Fanuc TP program (LS listing): makrostp.ls

/PROG  MAKROSTP
/ATTR
OWNER		= MNEDITOR;
COMMENT		= "MAKRO_SCHRITT";
PROG_SIZE	= 110862;
CREATE		= DATE 11-01-11  TIME 07:00:00;
MODIFIED	= DATE 18-04-15  TIME 10:51:52;
FILE_NAME	= ;
VERSION		= 0;
LINE_COUNT	= 4830;
MEMORY_SIZE	= 113490;
PROTECT		= READ_WRITE;
TCD:  STACK_SIZE	= 0,
      TASK_PRIORITY	= 100,
      TIME_SLICE	= 0,
      BUSY_LAMP_OFF	= 1,
      ABORT_REQUEST	= 7,
      PAUSE_REQUEST	= 3;
DEFAULT_GROUP	= *,*,*,*,*;
CONTROL_CODE	= 00000000 00000010;
/MN
   1:  !Schrittkette Konzernstandard ;
   2:  !KS24 ;
   3:  !Version: 02 ;
   4:  !Stand: 011 ;
   5:  !letzte Aenderung 22.03.2017 KN ;
   6:   ;
   7:  !Zaehler [41] = aktueller Schritt ;
   8:  !Zaehler [42] = letzter Schritt ;
   9:  R[41]=0    ;
  10:  R[42]=0    ;
  11:   ;
  12:   ;
  13:  !*********************** ;
  14:  !*********************** ;
  15:  !* Start Makro_Schritt * ;
  16:  !*********************** ;
  17:  !*********************** ;
  18:   ;
  19:   ;
  20:  !***************************** ;
  21:  !*         Schritt 1         * ;
  22:  !* E/A's / Flags Ruecksetzen * ;
  23:  !***************************** ;
  24:   ;
  25:  !Loop fuer Schrittkette LBL[1] ;
  26:  LBL[1] ;
  27:  R[41]=1    ;
  28:  !Statusbildschirm einblenden ;
  29:  DO[18181]=(OFF) ;
  30:  !SK1 KF1 KS1 KE1 ;
  31:  DO[786]=(F[830] AND DO[786]) ;
  32:  DO[722]=(!F[830] AND DO[722]) ;
  33:  DO[834]=(OFF) ;
  34:  DO[842]=(OFF) ;
  35:  DO[847]=(OFF) ;
  36:  !SK2 KF2 KS2 KE2 ;
  37:  DO[946]=(F[831] AND DO[946]) ;
  38:  DO[882]=(!F[831] AND DO[882]) ;
  39:  DO[994]=(OFF) ;
  40:  DO[995]=(OFF) ;
  41:  DO[1002]=(OFF) ;
  42:  !SK3 KF3 KS3 KE3 ;
  43:  DO[1106]=(F[832] AND DO[1106]) ;
  44:  DO[1042]=(!F[832] AND DO[1042]) ;
  45:  DO[1154]=(OFF) ;
  46:  DO[1155]=(OFF) ;
  47:  DO[1162]=(OFF) ;
  48:  !KS1 KS2 KS3 ;
  49:  DO[3969]=(OFF) ;
  50:  DO[3970]=(OFF) ;
  51:  DO[3971]=(OFF) ;
  52:  !Auswahl EZ1/SP1 an KF2 ;
  53:  F[72]=(OFF) ;
  54:  !Auswahl EZ1/SP1 an KF3 ;
  55:  F[73]=(OFF) ;
  56:  !Auswert. KF Umdrehungen EZ1/SP1 ;
  57:  F[94]=(OFF) ;
  58:  F[95]=(OFF) ;
  59:  F[96]=(OFF) ;
  60:  F[97]=(OFF) ;
  61:  F[98]=(OFF) ;
  62:  F[99]=(OFF) ;
  63:  F[100]=(OFF) ;
  64:  F[101]=(OFF) ;
  65:  F[102]=(OFF) ;
  66:  F[103]=(OFF) ;
  67:  F[104]=(OFF) ;
  68:  F[105]=(OFF) ;
  69:  F[106]=(OFF) ;
  70:  F[107]=(OFF) ;
  71:  F[108]=(OFF) ;
  72:  F[109]=(OFF) ;
  73:  F[110]=(OFF) ;
  74:  F[111]=(OFF) ;
  75:  F[112]=(OFF) ;
  76:  F[113]=(OFF) ;
  77:  F[114]=(OFF) ;
  78:  F[115]=(OFF) ;
  79:  F[116]=(OFF) ;
  80:  F[117]=(OFF) ;
  81:  !Auswert. KF Umdrehungen EZ2/SP2 ;
  82:  F[150]=(OFF) ;
  83:  F[151]=(OFF) ;
  84:  F[152]=(OFF) ;
  85:  F[153]=(OFF) ;
  86:  F[154]=(OFF) ;
  87:  F[155]=(OFF) ;
  88:  !Auswert. KF Umdrehungen EZ3/SP3 ;
  89:  F[186]=(OFF) ;
  90:  F[187]=(OFF) ;
  91:  F[188]=(OFF) ;
  92:  F[189]=(OFF) ;
  93:  F[190]=(OFF) ;
  94:  F[191]=(OFF) ;
  95:  !Hilfsflags beim Fraesen ;
  96:  F[287]=(OFF) ;
  97:  F[290]=(OFF) ;
  98:  F[291]=(OFF) ;
  99:  F[301]=(OFF) ;
 100:  !Hilfsflags SZ2 an SK1 ;
 101:  F[307]=(OFF) ;
 102:  F[308]=(OFF) ;
 103:  !Hilfsflags KF Initiator ;
 104:  F[312]=(OFF) ;
 105:  F[313]=(OFF) ;
 106:  !RSK Fehlerausgaben ;
 107:  F[322]=(OFF) ;
 108:  F[323]=(OFF) ;
 109:  F[324]=(OFF) ;
 110:  F[325]=(OFF) ;
 111:  F[326]=(OFF) ;
 112:  F[327]=(OFF) ;
 113:  F[328]=(OFF) ;
 114:  F[329]=(OFF) ;
 115:  !Flag KL1 Spueleimer ;
 116:  F[352]=(OFF) ;
 117:  F[353]=(OFF) ;
 118:  !Flag KL2 Spueleimer ;
 119:  F[373]=(OFF) ;
 120:  F[374]=(OFF) ;
 121:  !Flag KL3 Spueleimer ;
 122:  F[394]=(OFF) ;
 123:  F[395]=(OFF) ;
 124:  !Flag MS Reinigung gestartet ;
 125:  F[604]=(OFF) ;
 126:  F[605]=(OFF) ;
 127:  F[608]=(OFF) ;
 128:  !Flag für Grundstellung RSK ;
 129:  F[321]=(OFF) ;
 130:  !Ruecksetzen Fraeszaehler ;
 131:  R[1]=0    ;
 132:  R[42]=1    ;
 133:  JMP LBL[2] ;
 134:   ;
 135:   ;
 136:  !************************ ;
 137:  !************************ ;
 138:  !* RSK in Grundstellung * ;
 139:  !************************ ;
 140:  !************************ ;
 141:   ;
 142:   ;
 143:  !*********************** ;
 144:  !*      Schritt 2      * ;
 145:  !* Funktionsauswertung * ;
 146:  !*********************** ;
 147:   ;
 148:  LBL[2] ;
 149:  R[41]=2    ;
 150:  F[321]=(ON) ;
 151:   ;
 152:  !Fraesen ROB EZ1/SP1 SZ1-SZ4 ;
 153:  !an KF1 ;
 154:  IF ((F[90] AND !F[91]) AND !F[72] AND !F[73] AND !F[565] AND (F[64] OR F[65] OR F[66] OR F[67])),R[41]=3 ;
 155:   ;
 156:  !Fraesen ROB EZ1/SP1 SZ1-SZ4 ;
 157:  !an KF2 ;
 158:  IF ((F[90] AND !F[91]) AND F[72] AND !F[73] AND !F[565] AND (F[64] OR F[65] OR F[66] OR F[67])),R[41]=58 ;
 159:   ;
 160:  !Fraesen ROB EZ1/SP1 SZ1-SZ4 ;
 161:  !an KF3 ;
 162:  IF ((F[90] AND !F[91]) AND !F[72] AND F[73] AND !F[565] AND (F[64] OR F[65] OR F[66] OR F[67])),R[41]=64 ;
 163:   ;
 164:  !Fraesen STAT EZ1/SP1 ;
 165:  IF (F[92] AND !F[93]),R[41]=9 ;
 166:   ;
 167:  !Fraesen STAT EZ2/SP2 ;
 168:  IF (F[148] AND !F[149]),R[41]=18 ;
 169:   ;
 170:  !Fraesen STAT EZ3/SP3 ;
 171:  IF (F[184] AND !F[185]),R[41]=27 ;
 172:   ;
 173:  !MS1 Reinigung an KS3 ;
 174:  IF (F[603] AND !F[605] AND F[528] AND !F[529]),R[41]=36 ;
 175:   ;
 176:  !MS2 Reinigung an KS2 ;
 177:  IF (F[607] AND !F[609] AND F[528] AND !F[529]),R[41]=40 ;
 178:   ;
 179:  !KL1 Spueleimer (an Pneum. Schwen ;
 180:  !in Arbeitsstellung schwenken ;
 181:  IF (!F[352] AND F[353] AND !F[355] AND ((F[523] AND !F[524]) OR (!F[523] AND F[524]))),R[41]=44 ;
 182:   ;
 183:  !KL1 Spueleimer (an Pneum. Schwen ;
 184:  !in Ruhestellung schwenken ;
 185:  IF (F[352] AND !F[353] AND !F[355] AND ((F[523] AND !F[524]) OR (!F[523] AND F[524]))),R[41]=45 ;
 186:   ;
 187:  !KL2 Spueleimer (an Pneum. Schwen ;
 188:  !in Arbeitsstellung schwenken ;
 189:  IF (!F[373] AND F[374] AND !F[376] AND ((F[523] AND !F[524]) OR (!F[523] AND F[524]))),R[41]=46 ;
 190:   ;
 191:  !KL2 Spueleimer (an Pneum. Schwen ;
 192:  !in Ruhestellung schwenken ;
 193:  IF (F[373] AND !F[374] AND !F[376] AND ((F[523] AND !F[524]) OR (!F[523] AND F[524]))),R[41]=47 ;
 194:   ;
 195:  !KL3 Spueleimer (an Pneum. Schwen ;
 196:  !in Arbeitsstellung schwenken ;
 197:  IF (!F[394] AND F[395] AND !F[397] AND ((F[523] AND !F[524]) OR (!F[523] AND F[524]))),R[41]=48 ;
 198:   ;
 199:  !KL3 Spueleimer (an Pneum. Schwen ;
 200:  !in Ruhestellung schwenken ;
 201:  IF (F[394] AND !F[395] AND !F[397] AND ((F[523] AND !F[524]) OR (!F[523] AND F[524]))),R[41]=49 ;
 202:   ;
 203:  !MS1 Reinigung (an Pneum. Schwenk ;
 204:  IF (F[603] AND !F[605] AND !F[528] AND F[529]),R[41]=50 ;
 205:   ;
 206:  !Fraesen ROB STP SZ1 ;
 207:  IF (F[64] AND !F[65] AND !F[66] AND !F[67] AND F[90] AND !F[91] AND F[565] AND !F[805]),R[41]=70 ;
 208:   ;
 209:  !Fraesen ROB STP SZ1 mit Kappenw. ;
 210:  IF (F[64] AND !F[65] AND !F[66] AND !F[67] AND F[90] AND !F[91] AND F[565] AND F[805]),R[41]=76 ;
 211:   ;
 212:  !Warte Zeit für CPU ;
 213:  WAIT    .20(sec) ;
 214:   ;
 215:  R[42]=2    ;
 216:  JMP LBL[R[41]] ;
 217:   ;
 218:   ;
 219:  !*************************** ;
 220:  !*************************** ;
 221:  !* Fraesen Rob EZ1 SZ1-SZ4 * ;
 222:  !*          an KF1         * ;
 223:  !*************************** ;
 224:  !*************************** ;
 225:   ;
 226:   ;
 227:  !**************************** ;
 228:  !*        Schritt 3         * ;
 229:  !* Rob EZ1 SZ1-SZ4 Auswert. * ;
 230:  !**************************** ;
 231:   ;
 232:  LBL[3] ;
 233:  R[41]=3    ;
 234:  !RSK gestartet ;
 235:  F[321]=(OFF) ;
 236:  GO[1]=(31) ;
 237:  IF (F[64]),GO[3]=(31) ;
 238:  IF (F[65]),GO[3]=(32) ;
 239:  IF (F[66]),GO[3]=(33) ;
 240:  IF (F[67]),GO[3]=(34) ;
 241:  WAIT    .10(sec) ;
 242:  DO[116]=(ON) ;
 243:  DO[130]=(ON) ;
 244:  DO[718]=(OFF) ;
 245:  DO[717]=(!DI[717]) ;
 246:  DO[18181]=(ON) ;
 247:  WAIT (DI[717])    ;
 248:  DO[18181]=(OFF) ;
 249:  DO[717]=(OFF) ;
 250:  !Anwahl Startfraesen ;
 251:  IF (F[90] AND F[78] AND !F[79]),R[41]=4 ;
 252:  !Anwahl Normalfraesen ;
 253:  IF (F[90] AND !F[78] AND F[79]),R[41]=6 ;
 254:  R[42]=3    ;
 255:  JMP LBL[R[41]] ;
 256:   ;
 257:  !***************************** ;
 258:  !*         Schritt 4         * ;
 259:  !* Rob EZ1 SZ1-SZ4 SF Teil 1 * ;
 260:  !***************************** ;
 261:   ;
 262:  LBL[4] ;
 263:  R[41]=4    ;
 264:  !RSK gestartet ;
 265:  F[321]=(OFF) ;
 266:  F[329]=(OFF) ;
 267:  F[325]=(OFF) ;
 268:  DO[718]=(OFF) ;
 269:  DO[717]=(!DI[717]) ;
 270:  DO[18181]=(ON) ;
 271:  WAIT (DI[717])    ;
 272:  DO[18181]=(OFF) ;
 273:  DO[834]=(ON) ;
 274:  DO[858]=(ON) ;
 275:  DO[835]=(F[330]) ;
 276:  DO[859]=(F[330]) ;
 277:  DO[717]=(OFF) ;
 278:  !Warte Fraeser laeuft ;
 279:  TIMER[7]=((-3)) ;
 280:  WAIT ((!DI[834] AND !F[289]) OR (!DI[858] AND F[289]) OR (TIMER[7]>=0))    ;
 281:  WAIT ((DI[834] AND !F[289]) OR (DI[858] AND F[289]) OR (TIMER[7]>=0))    ;
 282:  F[322]=((TIMER[7]>=0)) ;
 283:  DO[18181]=(ON) ;
 284:  WAIT ((!DI[834] AND !F[289]) OR (!DI[858] AND F[289]))    ;
 285:  WAIT ((DI[834] AND !F[289]) OR (DI[858] AND F[289]))    ;
 286:  DO[18181]=(OFF) ;
 287:  F[322]=(OFF) ;
 288:  !EZ1/SP1 schliessen ;
 289:  DO[718]=(ON) ;
 290:  TIMER[9]=((-4)) ;
 291:  !EZ1/SP1 Kraft erreicht ;
 292:  WAIT ((DI[718] AND !DI[772] AND !DI[780] AND !DI[774] AND !DI[775]) OR (TIMER[9]>=0))    ;
 293:  DO[18181]=(ON) ;
 294:  DO[718]=((TIMER[9]<0)) ;
 295:  DO[834]=((TIMER[9]<0)) ;
 296:  DO[858]=((TIMER[9]<0)) ;
 297:  WAIT ((DI[718] AND !DI[772] AND !DI[780] AND !DI[774] AND !DI[775]) OR DI[26] OR DI[27])    ;
 298:  F[325]=(DI[26] OR DI[27]) ;
 299:  DO[18181]=(OFF) ;
 300:  !EZ1/SP1 Fehler Kraftaufbau ;
 301:  IF (F[325]),JMP LBL[406] ;
 302:  TIMER[9]=((-5)) ;
 303:  LBL[400] ;
 304:  WAIT ((!DI[834] AND !F[289]) OR (!DI[858] AND F[289]) OR F[325] OR (TIMER[9]>=0))    ;
 305:  WAIT ((DI[834] AND !F[289]) OR (DI[858] AND F[289]) OR F[325] OR (TIMER[9]>=0))    ;
 306:  R[1]=(R[1]+1) ;
 307:  F[329]=((TIMER[9]>=0)) ;
 308:  !Fraeszeit ueberschritten ;
 309:  IF (F[329]),JMP LBL[406] ;
 310:  IF (F[64]),JMP LBL[402] ;
 311:  IF (F[65]),JMP LBL[403] ;
 312:  IF (F[66]),JMP LBL[404] ;
 313:  IF (F[67]),JMP LBL[405] ;
 314:  !Umdrehungen Vergl.SZ1 ;
 315:  LBL[402] ;
 316:  !Umdrehungen Vergleichen ;
 317:  IF (R[1]<R[2]),JMP LBL[400] ;
 318:  JMP LBL[401] ;
 319:  !Umdrehungen Vergl.SZ2 ;
 320:  LBL[403] ;
 321:  !Umdrehungen Vergleichen ;
 322:  IF (R[1]<R[8]),JMP LBL[400] ;
 323:  JMP LBL[401] ;
 324:  !Umdrehungen Vergl.SZ3 ;
 325:  LBL[404] ;
 326:  !Umdrehungen Vergleichen ;
 327:  IF (R[1]<R[11]),JMP LBL[400] ;
 328:  JMP LBL[401] ;
 329:  !Umdrehungen Vergl.SZ4 ;
 330:  LBL[405] ;
 331:  !Umdrehungen Vergleichen ;
 332:  IF (R[1]<R[14]),JMP LBL[400] ;
 333:  JMP LBL[401] ;
 334:  LBL[401] ;
 335:  IF (F[64]),F[94]=(ON) ;
 336:  IF (F[65]),F[100]=(ON) ;
 337:  IF (F[66]),F[106]=(ON) ;
 338:  IF (F[67]),F[112]=(ON) ;
 339:  LBL[406] ;
 340:  DO[834]=((TIMER[9]<0)) ;
 341:  DO[858]=((TIMER[9]<0)) ;
 342:  !Fraeser ausblasen EIN ;
 343:  DO[835]=(F[330] OR (TIMER[9]<0)) ;
 344:  DO[859]=(F[330] OR (TIMER[9]<0)) ;
 345:  DO[718]=(OFF) ;
 346:  !EZ1/SP1 oeffnen ;
 347:  DO[717]=(!DI[717]) ;
 348:  DO[18181]=(F[329]) ;
 349:  WAIT (!F[329] OR DI[26] OR DI[27])    ;
 350:  DO[18181]=(OFF) ;
 351:  DO[18181]=(ON) ;
 352:  WAIT (DI[717])    ;
 353:  DO[18181]=(OFF) ;
 354:  DO[717]=(OFF) ;
 355:  !Umdrehungen ruecksetzen ;
 356:  R[1]=0    ;
 357:  R[42]=4    ;
 358:  IF (F[329] OR F[325]),JMP LBL[4] ;
 359:  JMP LBL[5] ;
 360:   ;
 361:  !***************************** ;
 362:  !*         Schritt 5         * ;
 363:  !* Rob EZ1 SZ1-SZ4 SF Teil 2 * ;
 364:  !***************************** ;
 365:   ;
 366:  LBL[5] ;
 367:  R[41]=5    ;
 368:  !RSK gestartet ;
 369:  F[321]=(OFF) ;
 370:  F[329]=(OFF) ;
 371:  F[325]=(OFF) ;
 372:  DO[718]=(OFF) ;
 373:  DO[717]=(!DI[717]) ;
 374:  DO[18181]=(ON) ;
 375:  WAIT (DI[717])    ;
 376:  DO[18181]=(OFF) ;
 377:  DO[834]=(ON) ;
 378:  DO[858]=(ON) ;
 379:  DO[717]=(OFF) ;
 380:  !EZ1/SP1 schliessen ;
 381:  DO[718]=(ON) ;
 382:  !Fraeser ausblasen AUS/AN ;
 383:  DO[835]=(F[330]) ;
 384:  DO[859]=(F[330]) ;
 385:  TIMER[9]=((-4)) ;
 386:  !EZ1/SP1 Kraft erreicht ;
 387:  WAIT ((DI[718] AND !DI[772] AND !DI[780] AND !DI[774] AND !DI[775]) OR (TIMER[9]>=0))    ;
 388:  DO[18181]=(ON) ;
 389:  DO[718]=((TIMER[9]<0)) ;
 390:  DO[834]=((TIMER[9]<0)) ;
 391:  DO[858]=((TIMER[9]<0)) ;
 392:  WAIT ((DI[718] AND !DI[772] AND !DI[780] AND !DI[774] AND !DI[775]) OR DI[26] OR DI[27])    ;
 393:  F[325]=(DI[26] OR DI[27]) ;
 394:  DO[18181]=(OFF) ;
 395:  !EZ1/SP1 Fehler Kraftaufbau ;
 396:  IF (F[325]),JMP LBL[5] ;
 397:  TIMER[9]=((-5)) ;
 398:  LBL[500] ;
 399:  WAIT ((!DI[834] AND !F[289]) OR (!DI[858] AND F[289]) OR F[325] OR (TIMER[9]>=0))    ;
 400:  WAIT ((DI[834] AND !F[289]) OR (DI[858] AND F[289]) OR F[325] OR (TIMER[9]>=0))    ;
 401:  R[1]=(R[1]+1) ;
 402:  F[329]=((TIMER[9]>=0)) ;
 403:  !Fraeszeit ueberschritten ;
 404:  IF (F[329]),JMP LBL[506] ;
 405:  IF (F[64]),JMP LBL[502] ;
 406:  IF (F[65]),JMP LBL[503] ;
 407:  IF (F[66]),JMP LBL[504] ;
 408:  IF (F[67]),JMP LBL[505] ;
 409:  !Umdrehungen Vergl.SZ1 ;
 410:  LBL[502] ;
 411:  !Umdrehungen Vergleichen ;
 412:  IF (R[1]<R[3]),JMP LBL[500] ;
 413:  JMP LBL[501] ;
 414:  !Umdrehungen Vergl.SZ2 ;
 415:  LBL[503] ;
 416:  !Umdrehungen Vergleichen ;
 417:  IF (R[1]<R[9]),JMP LBL[500] ;
 418:  JMP LBL[501] ;
 419:  !Umdrehungen Vergl.SZ3 ;
 420:  LBL[504] ;
 421:  !Umdrehungen Vergleichen ;
 422:  IF (R[1]<R[12]),JMP LBL[500] ;
 423:  JMP LBL[501] ;
 424:  !Umdrehungen Vergl.SZ4 ;
 425:  LBL[505] ;
 426:  !Umdrehungen Vergleichen ;
 427:  IF (R[1]<R[15]),JMP LBL[500] ;
 428:  JMP LBL[501] ;
 429:  LBL[501] ;
 430:  IF (F[64]),F[96]=(ON) ;
 431:  IF (F[65]),F[102]=(ON) ;
 432:  IF (F[66]),F[108]=(ON) ;
 433:  IF (F[67]),F[114]=(ON) ;
 434:  LBL[506] ;
 435:  DO[834]=((TIMER[9]<0)) ;
 436:  DO[858]=((TIMER[9]<0)) ;
 437:  !Fraeser ausblasen EIN ;
 438:  DO[835]=PULSE,4.0sec ;
 439:  DO[859]=PULSE,4.0sec ;
 440:  DO[718]=(OFF) ;
 441:  !EZ1/SP1 oeffnen ;
 442:  DO[717]=(!DI[717]) ;
 443:  DO[18181]=(F[329]) ;
 444:  WAIT (!F[329] OR DI[26] OR DI[27])    ;
 445:  DO[18181]=(OFF) ;
 446:  DO[18181]=(ON) ;
 447:  WAIT (DI[717])    ;
 448:  DO[18181]=(OFF) ;
 449:  DO[717]=(OFF) ;
 450:  !Umdrehungen ruecksetzen ;
 451:  R[1]=0    ;
 452:  R[42]=5    ;
 453:  IF (F[329] OR F[325]),JMP LBL[5] ;
 454:  JMP LBL[7] ;
 455:   ;
 456:  !********************** ;
 457:  !*     Schritt 6      * ;
 458:  !* Rob EZ1 SZ1-SZ4 NF * ;
 459:  !********************** ;
 460:   ;
 461:  LBL[6] ;
 462:  R[41]=6    ;
 463:  !RSK gestartet ;
 464:  F[321]=(OFF) ;
 465:  F[329]=(OFF) ;
 466:  F[325]=(OFF) ;
 467:  !Zähler wegspeichern für 2ten Hub ;
 468:  R[45]=(R[4]) ;
 469:  IF (F[98] AND F[732]),R[4]=(R[43]) ;
 470:  !Überprüfungung Zangenstellung ;
 471:  DO[718]=(OFF) ;
 472:  DO[717]=(!DI[717]) ;
 473:  DO[18181]=(ON) ;
 474:  WAIT (DI[717])    ;
 475:  DO[18181]=(OFF) ;
 476:  DO[834]=(ON) ;
 477:  DO[835]=(F[330]) ;
 478:  DO[858]=(ON) ;
 479:  DO[859]=(F[330]) ;
 480:  DO[717]=(OFF) ;
 481:  !Warte Fraeser laeuft ;
 482:  TIMER[7]=((-3)) ;
 483:  WAIT ((!DI[834] AND !F[289]) OR (!DI[858] AND F[289]) OR (TIMER[7]>=0))    ;
 484:  WAIT ((DI[834] AND !F[289]) OR (DI[858] AND F[289]) OR (TIMER[7]>=0))    ;
 485:  F[322]=((TIMER[7]>=0)) ;
 486:  DO[18181]=(ON) ;
 487:  WAIT ((!DI[834] AND !F[289]) OR (!DI[858] AND F[289]))    ;
 488:  WAIT ((DI[834] AND !F[289]) OR (DI[858] AND F[289]))    ;
 489:  DO[18181]=(OFF) ;
 490:  F[322]=(OFF) ;
 491:  !EZ1/SP1 schliessen ;
 492:  DO[718]=(ON) ;
 493:  TIMER[9]=((-4)) ;
 494:  !EZ1/SP1 Kraft erreicht ;
 495:  WAIT ((DI[718] AND !DI[772] AND !DI[780] AND !DI[774] AND !DI[775]) OR (TIMER[9]>=0))    ;
 496:  DO[18181]=(ON) ;
 497:  DO[718]=((TIMER[9]<0)) ;
 498:  DO[834]=((TIMER[9]<0)) ;
 499:  DO[858]=((TIMER[9]<0)) ;
 500:  WAIT ((DI[718] AND !DI[772] AND !DI[780] AND !DI[774] AND !DI[775]) OR DI[26] OR DI[27])    ;
 501:  F[325]=(DI[26] OR DI[27]) ;
 502:  DO[18181]=(OFF) ;
 503:  !EZ1/SP1 Fehler Kraftaufbau ;
 504:  IF (F[325]),JMP LBL[6] ;
 505:  TIMER[9]=((-5)) ;
 506:  LBL[600] ;
 507:  WAIT ((!DI[834] AND !F[289]) OR (!DI[858] AND F[289]) OR F[325] OR (TIMER[9]>=0))    ;
 508:  WAIT ((DI[834] AND !F[289]) OR (DI[858] AND F[289]) OR F[325] OR (TIMER[9]>=0))    ;
 509:  R[1]=(R[1]+1) ;
 510:  F[329]=((TIMER[9]>=0)) ;
 511:  !Fraeszeit ueberschritten ;
 512:  IF (F[329]),JMP LBL[606] ;
 513:  IF (F[64]),JMP LBL[602] ;
 514:  IF (F[65]),JMP LBL[603] ;
 515:  IF (F[66]),JMP LBL[604] ;
 516:  IF (F[67]),JMP LBL[605] ;
 517:  !Umdrehungen Vergl.SZ1 ;
 518:  LBL[602] ;
 519:  !Umdrehungen Vergleichen ;
 520:  IF (R[1]<R[4]),JMP LBL[600] ;
 521:  JMP LBL[601] ;
 522:  !Umdrehungen Vergl.SZ2 ;
 523:  LBL[603] ;
 524:  !Umdrehungen Vergleichen ;
 525:  IF (R[1]<R[10]),JMP LBL[600] ;
 526:  !Umdrehungen Vergl.SZ3 ;
 527:  LBL[604] ;
 528:  !Umdrehungen Vergleichen ;
 529:  IF (R[1]<R[13]),JMP LBL[600] ;
 530:  JMP LBL[601] ;
 531:  !Umdrehungen Vergl.SZ4 ;
 532:  LBL[605] ;
 533:  !Umdrehungen Vergleichen ;
 534:  IF (R[1]<R[16]),JMP LBL[600] ;
 535:  LBL[601] ;
 536:  !EZ1/SP1 2 Huebe bei NF ;
 537:  IF (!F[130]),JMP LBL[606] ;
 538:  IF (F[98]),F[96]=(ON) ;
 539:  IF (F[104]),F[96]=(ON) ;
 540:  IF (F[110]),F[96]=(ON) ;
 541:  IF (F[116]),F[96]=(ON) ;
 542:  IF (F[64]),F[98]=(ON) ;
 543:  IF (F[65]),F[104]=(ON) ;
 544:  IF (F[66]),F[110]=(ON) ;
 545:  IF (F[67]),F[116]=(ON) ;
 546:  LBL[606] ;
 547:  DO[834]=((TIMER[9]<0)) ;
 548:  DO[858]=((TIMER[9]<0)) ;
 549:  !Fraeser ausblasen EIN ;
 550:  DO[835]=PULSE,4.0sec ;
 551:  DO[859]=PULSE,4.0sec ;
 552:  DO[718]=(OFF) ;
 553:  !EZ1/SP1 oeffnen ;
 554:  DO[717]=(!DI[717]) ;
 555:  DO[18181]=(F[329]) ;
 556:  WAIT (!F[329] OR DI[26] OR DI[27])    ;
 557:  DO[18181]=(OFF) ;
 558:  DO[18181]=(ON) ;
 559:  WAIT (DI[717])    ;
 560:  DO[18181]=(OFF) ;
 561:  DO[717]=(OFF) ;
 562:  !Umdrehungen ruecksetzen ;
 563:  R[1]=0    ;
 564:  R[42]=6    ;
 565:  !Zähler umschreiben für 2ten Hub ;
 566:  IF (F[98] AND F[732] AND F[64]),GO[3]=36 ;
 567:  IF (F[104] AND F[732] AND F[65]),GO[3]=37 ;
 568:  IF (F[110] AND F[732] AND F[66]),GO[3]=38 ;
 569:  IF (F[116] AND F[732] AND F[67]),GO[3]=39 ;
 570:  IF (F[96] AND F[732]),R[4]=(R[45]) ;
 571:  !Aufruf 2ter Hub ;
 572:  IF (F[329] OR (!F[96] AND F[130])),JMP LBL[6] ;
 573:  IF (F[64]),F[98]=(ON) ;
 574:  IF (F[65]),F[104]=(ON) ;
 575:  IF (F[66]),F[110]=(ON) ;
 576:  IF (F[67]),F[116]=(ON) ;
 577:  JMP LBL[7] ;
 578:   ;
 579:  !******************************* ;
 580:  !*         Schritt 7           * ;
 581:  !* Rob EZ1 SZ1-SZ4 i.O./n.i.O. * ;
 582:  !******************************* ;
 583:   ;
 584:  LBL[7] ;
 585:  R[41]=7    ;
 586:  !Fraesueberwachung starten ;
 587:  IF (F[64]),JMP LBL[701] ;
 588:  IF (F[65]),JMP LBL[702] ;
 589:  IF (F[66]),JMP LBL[703] ;
 590:  IF (F[67]),JMP LBL[704] ;
 591:  LBL[701] ;
 592:  TIMER[7]=((-3)) ;
 593:  WAIT (F[64] AND ((F[79] AND F[98]) OR (F[78] AND F[94] AND F[96])) OR (TIMER[7]>=0))    ;
 594:  F[329]=((TIMER[7]>=0)) ;
 595:  DO[18181]=(ON) ;
 596:  WAIT (F[64] AND ((F[79] AND F[98]) OR (F[78] AND F[94] AND F[96])))    ;
 597:  DO[18181]=(OFF) ;
 598:  JMP LBL[700] ;
 599:  LBL[702] ;
 600:  TIMER[7]=((-3)) ;
 601:  WAIT (F[65] AND ((F[79] AND F[104]) OR (F[78] AND F[100] AND F[102])) OR (TIMER[7]>=0))    ;
 602:  F[329]=((TIMER[7]>=0)) ;
 603:  DO[18181]=(ON) ;
 604:  WAIT (F[65] AND ((F[79] AND F[104]) OR (F[78] AND F[100] AND F[102])))    ;
 605:  DO[18181]=(OFF) ;
 606:  JMP LBL[700] ;
 607:  LBL[703] ;
 608:  TIMER[7]=((-3)) ;
 609:  WAIT (F[66] AND ((F[79] AND F[110]) OR (F[78] AND F[106] AND F[108])) OR (TIMER[7]>=0))    ;
 610:  F[329]=((TIMER[7]>=0)) ;
 611:  DO[18181]=(ON) ;
 612:  WAIT (F[66] AND ((F[79] AND F[110]) OR (F[78] AND F[106] AND F[108])))    ;
 613:  DO[18181]=(OFF) ;
 614:  JMP LBL[700] ;
 615:  LBL[704] ;
 616:  TIMER[7]=((-3)) ;
 617:  WAIT (F[67] AND ((F[79] AND F[116]) OR (F[78] AND F[112] AND F[114])) OR (TIMER[7]>=0))    ;
 618:  F[329]=((TIMER[7]>=0)) ;
 619:  DO[18181]=(ON) ;
 620:  WAIT (F[67] AND ((F[79] AND F[116]) OR (F[78] AND F[112] AND F[114])))    ;
 621:  DO[18181]=(OFF) ;
 622:  JMP LBL[700] ;
 623:  LBL[700] ;
 624:  R[41]=8    ;
 625:  !KF1 U-Merker ruecksetzen ;
 626:  F[94]=(OFF) ;
 627:  F[96]=(OFF) ;
 628:  F[98]=(OFF) ;
 629:  F[100]=(OFF) ;
 630:  F[102]=(OFF) ;
 631:  F[104]=(OFF) ;
 632:  F[106]=(OFF) ;
 633:  F[108]=(OFF) ;
 634:  F[110]=(OFF) ;
 635:  F[112]=(OFF) ;
 636:  F[114]=(OFF) ;
 637:  F[116]=(OFF) ;
 638:  R[42]=7    ;
 639:  JMP LBL[R[41]] ;
 640:   ;
 641:  !***************************** ;
 642:  !*        Schritt 8          * ;
 643:  !* Rob EZ1 SZ1-SZ4 Quitt SK1 * ;
 644:  !* Rob EZ1 SZ1-SZ4 Quitt KE1 * ;
 645:  !***************************** ;
 646:   ;
 647:  LBL[8] ;
 648:  R[41]=8    ;
 649:  !RSK gestartet ;
 650:  F[321]=(OFF) ;
 651:  IF (F[64]),GO[3]=1 ;
 652:  IF (F[65]),GO[3]=2 ;
 653:  IF (F[66]),GO[3]=3 ;
 654:  IF (F[67]),GO[3]=4 ;
 655:  WAIT    .10(sec) ;
 656:  DO[786]=(!F[830]) ;
 657:  DO[722]=(F[830]) ;
 658:  DO[116]=(OFF) ;
 659:  DO[130]=(OFF) ;
 660:  DO[18181]=(ON) ;
 661:  WAIT ((!DI[786] AND DI[787] AND !DI[788]) OR F[830])    ;
 662:  WAIT ((!DI[722] AND DI[724] AND !DI[723] OR F[329]) OR !F[830])    ;
 663:  !FK Fraesen ;
 664:  F[91]=((!DI[786] AND DI[787] AND !DI[788] AND !F[830]) OR (!DI[722] AND DI[724] AND !DI[723] AND F[830]) AND !F[322] AND !F[325] AND !F[329]) ;
 665:  DO[18181]=(OFF) ;
 666:  DO[786]=(F[830] AND DO[786]) ;
 667:  DO[722]=(!F[830] AND DO[722]) ;
 668:  R[42]=8    ;
 669:  JMP LBL[1] ;
 670:   ;
 671:   ;
 672:  !************************ ;
 673:  !************************ ;
 674:  !* Fraesen STAT EZ1/SP1 * ;
 675:  !************************ ;
 676:  !************************ ;
 677:   ;
 678:   ;
 679:  !****************************** ;
 680:  !*         Schritt 9          * ;
 681:  !*        STAT EZ1/SP1        * ;
 682:  !* KS1 in Arbeitsst.schwenken * ;
 683:  !****************************** ;
 684:   ;
 685:  LBL[9] ;
 686:  R[41]=9    ;
 687:  !RSK gestartet ;
 688:  F[321]=(OFF) ;
 689:  GO[1]=(31) ;
 690:  GO[3]=(31) ;
 691:  WAIT    .10(sec) ;
 692:  DO[758]=(F[78]) ;
 693:  DO[759]=(F[79]) ;
 694:  DO[116]=(ON) ;
 695:  DO[130]=(ON) ;
 696:  DO[718]=(OFF) ;
 697:  DO[717]=(!DI[717]) ;
 698:  DO[18181]=(ON) ;
 699:  WAIT (DI[717])    ;
 700:  DO[18181]=(OFF) ;
 701:  DO[717]=(OFF) ;
 702:  !Ueberwachungszeit Grundstellung ;
 703:  TIMER[8]=((-4)) ;
 704:  WAIT ((DI[842] AND !DI[843] AND !DI[844] AND DI[845]) OR (TIMER[8]>=0))    ;
 705:  F[323]=((TIMER[8]>=0)) ;
 706:  DO[18181]=((TIMER[8]>=0)) ;
 707:  WAIT (DI[842] AND !DI[843] AND !DI[844] AND DI[845])    ;
 708:  DO[18181]=(OFF) ;
 709:  F[323]=(OFF) ;
 710:  TIMER[8]=((-4)) ;
 711:  DO[835]=(F[564]) ;
 712:  WAIT ((DI[835] AND F[564]) OR (!DI[835] AND !F[564]) OR (TIMER[8]>=0))    ;
 713:  F[323]=((TIMER[8]>=0)) ;
 714:  DO[18181]=((TIMER[8]>=0)) ;
 715:  WAIT ((DI[835] AND F[564]) OR (!DI[835] AND !F[564]))    ;
 716:  DO[18181]=(OFF) ;
 717:  F[323]=(OFF) ;
 718:  !Ueberwachungszeit KS1 Schwenken ;
 719:  TIMER[8]=((-6)) ;
 720:  !KS1 in Arbeitst. schwenken ;
 721:  DO[3972]=(ON) ;
 722:  WAIT (DI[841] OR (TIMER[8]>=0))    ;
 723:  DO[18181]=((TIMER[8]>=0)) ;
 724:  WAIT (DI[841])    ;
 725:  TIMER[8]=((-6)) ;
 726:  DO[18181]=(OFF) ;
 727:  WAIT ((!DI[842] AND DI[843] AND DI[844] AND !DI[845]) OR (TIMER[8]>=0))    ;
 728:  F[324]=((TIMER[8]>=0)) ;
 729:  DO[3972]=(OFF) ;
 730:  DO[18181]=((TIMER[8]>=0)) ;
 731:  WAIT ((!DI[842] AND DI[843] AND DI[844] AND !DI[845]) OR DI[26])    ;
 732:  DO[18181]=(OFF) ;
 733:  F[324]=(OFF) ;
 734:  !Sprung zurueck bei KS1 Fehler ;
 735:  IF (TIMER[8]>=0),JMP LBL[9] ;
 736:  DO[835]=(OFF) ;
 737:  TIMER[11]=((R[24])) ;
 738:  WAIT ((TIMER[11]>=0) OR !F[564])    ;
 739:  TIMER[11]=STOP ;
 740:  DO[18181]=(ON) ;
 741:  WAIT ((F[92] AND F[78]) OR (F[92] AND F[79]))    ;
 742:  DO[18181]=(OFF) ;
 743:  !Anwahl Startfraesen ;
 744:  IF (!DI[842] AND DI[843] AND F[92] AND F[78] AND !F[301]),R[41]=10 ;
 745:  !Anwahl Normalfraesen ;
 746:  IF (!DI[842] AND DI[843] AND F[92] AND (F[79] OR F[301])),R[41]=12 ;
 747:  R[42]=9    ;
 748:  JMP LBL[R[41]] ;
 749:   ;
 750:  !************************** ;
 751:  !*       Schritt 10       * ;
 752:  !* STAT EZ1/SP1 SF Teil 1 * ;
 753:  !************************** ;
 754:   ;
 755:  LBL[10] ;
 756:  R[41]=10    ;
 757:  !RSK gestartet ;
 758:  F[321]=(OFF) ;
 759:  F[329]=(OFF) ;
 760:  F[325]=(OFF) ;
 761:  DO[718]=(OFF) ;
 762:  DO[717]=(!DI[717]) ;
 763:  DO[18181]=(ON) ;
 764:  WAIT (DI[717])    ;
 765:  DO[717]=(OFF) ;
 766:  DO[18181]=(OFF) ;
 767:  DO[834]=(ON) ;
 768:  !Warte Fraeser laeuft ;
 769:  TIMER[7]=((-3)) ;
 770:  WAIT (!DI[834] OR (TIMER[7]>=0))    ;
 771:  WAIT (DI[834] OR (TIMER[7]>=0))    ;
 772:  F[322]=((TIMER[7]>=0)) ;
 773:  DO[18181]=(ON) ;
 774:  WAIT (!DI[834])    ;
 775:  WAIT (DI[834])    ;
 776:  DO[18181]=(OFF) ;
 777:  F[322]=(OFF) ;
 778:  !EZ1/SP1 schliessen ;
 779:  DO[718]=(ON) ;
 780:  !Fraeser ausblasen AUS/EIN ;
 781:  DO[847]=(F[330]) ;
 782:  TIMER[9]=((-4)) ;
 783:  !EZ1/SP1 Kraft erreicht ;
 784:  WAIT ((DI[718] AND !DI[772] AND !DI[780] AND !DI[774] AND !DI[775]) OR (TIMER[9]>=0))    ;
 785:  F[325]=((TIMER[9]>=0)) ;
 786:  DO[18181]=(ON) ;
 787:  DO[718]=((TIMER[9]<0)) ;
 788:  DO[834]=((TIMER[9]<0)) ;
 789:  WAIT ((DI[718] AND !DI[772] AND !DI[780] AND !DI[774] AND !DI[775]) OR DI[26] OR DI[27])    ;
 790:  DO[18181]=(OFF) ;
 791:  !EZ1/SP1 Fehler Kraftaufbau ;
 792:  IF (F[325]),JMP LBL[1001] ;
 793:  TIMER[9]=((-5)) ;
 794:  LBL[1000] ;
 795:  WAIT (!DI[834] OR F[325] OR (TIMER[9]>=0))    ;
 796:  WAIT (DI[834] OR F[325] OR (TIMER[9]>=0))    ;
 797:  R[1]=(R[1]+1) ;
 798:  F[329]=((TIMER[9]>=0)) ;
 799:  !Fraeszeit ueberschritten ;
 800:  IF (F[329]),JMP LBL[1001] ;
 801:  !Umdrehungen Vergleichen ;
 802:  IF (R[1]<R[2]),JMP LBL[1000] ;
 803:  F[94]=(ON) ;
 804:  LBL[1001] ;
 805:  DO[834]=((TIMER[9]<0)) ;
 806:  !Fraeser ausblasen EIN ;
 807:  DO[847]=(F[330] OR (TIMER[9]<0)) ;
 808:  DO[718]=(OFF) ;
 809:  !EZ1/SP1 oeffnen ;
 810:  DO[717]=(!DI[717]) ;
 811:  DO[18181]=(F[329]) ;
 812:  WAIT (!F[329] OR DI[26] OR DI[27])    ;
 813:  DO[18181]=(OFF) ;
 814:  DO[18181]=(ON) ;
 815:  WAIT (DI[717])    ;
 816:  DO[18181]=(OFF) ;
 817:  DO[717]=(OFF) ;
 818:  !Umdrehungen ruecksetzen ;
 819:  R[1]=0    ;
 820:  R[42]=10    ;
 821:  IF (F[329] OR F[325]),JMP LBL[10] ;
 822:  JMP LBL[11] ;
 823:   ;
 824:  !************************** ;
 825:  !*       Schritt 11       * ;
 826:  !* STAT EZ1/SP1 SF Teil 2 * ;
 827:  !************************** ;
 828:   ;
 829:  LBL[11] ;
 830:  R[41]=11    ;
 831:  !RSK gestartet ;
 832:  F[321]=(OFF) ;
 833:  F[329]=(OFF) ;
 834:  F[325]=(OFF) ;
 835:  DO[718]=(OFF) ;
 836:  DO[717]=(!DI[717]) ;
 837:  DO[18181]=(ON) ;
 838:  WAIT (DI[717])    ;
 839:  DO[18181]=(OFF) ;
 840:  DO[834]=(ON) ;
 841:  DO[717]=(OFF) ;
 842:  !EZ1/SP1 schliessen ;
 843:  DO[718]=(ON) ;
 844:  !Fraeser ausblasen AUS/EIN ;
 845:  DO[847]=(F[330]) ;
 846:  TIMER[9]=((-4)) ;
 847:  !EZ1/SP1 Kraft erreicht ;
 848:  WAIT ((DI[718] AND !DI[772] AND !DI[780] AND !DI[774] AND !DI[775]) OR (TIMER[9]>=0))    ;
 849:  F[325]=((TIMER[9]>=0)) ;
 850:  DO[18181]=(ON) ;
 851:  DO[718]=((TIMER[9]<0)) ;
 852:  DO[834]=((TIMER[9]<0)) ;
 853:  WAIT ((DI[718] AND !DI[772] AND !DI[780] AND !DI[774] AND !DI[775]) OR DI[26] OR DI[27])    ;
 854:  DO[18181]=(OFF) ;
 855:  !EZ1/SP1 Fehler Kraftaufbau ;
 856:  IF (F[325]),JMP LBL[1101] ;
 857:  TIMER[9]=((-5)) ;
 858:  LBL[1100] ;
 859:  WAIT (!DI[834] OR F[325] OR (TIMER[9]>=0))    ;
 860:  WAIT (DI[834] OR F[325] OR (TIMER[9]>=0))    ;
 861:  R[1]=(R[1]+1) ;
 862:  F[329]=((TIMER[9]>=0)) ;
 863:  !Fraeszeit ueberschritten ;
 864:  IF (F[329]),JMP LBL[1101] ;
 865:  !Umdrehungen Vergleichen ;
 866:  IF (R[1]<R[3]),JMP LBL[1100] ;
 867:  F[96]=(ON) ;
 868:  LBL[1101] ;
 869:  DO[834]=((TIMER[9]<0)) ;
 870:  !Fraeser ausblasen EIN ;
 871:  DO[847]=PULSE,4.0sec ;
 872:  DO[718]=(OFF) ;
 873:  !EZ1/SP1 oeffnen ;
 874:  DO[717]=(!DI[717]) ;
 875:  DO[18181]=(F[329]) ;
 876:  WAIT (!F[329] OR DI[26] OR DI[27])    ;
 877:  DO[18181]=(OFF) ;
 878:  DO[18181]=(ON) ;
 879:  WAIT (DI[717])    ;
 880:  DO[18181]=(OFF) ;
 881:  DO[717]=(OFF) ;
 882:  !Umdrehungen ruecksetzen ;
 883:  R[1]=0    ;
 884:  R[42]=11    ;
 885:  IF (F[329] OR F[325]),JMP LBL[11] ;
 886:  JMP LBL[13] ;
 887:   ;
 888:  !******************* ;
 889:  !*   Schritt 12    * ;
 890:  !* STAT EZ1/SP1 NF * ;
 891:  !******************* ;
 892:   ;
 893:  LBL[12] ;
 894:  R[41]=12    ;
 895:  !RSK gestartet ;
 896:  F[321]=(OFF) ;
 897:  F[329]=(OFF) ;
 898:  F[325]=(OFF) ;
 899:  !Zähler wegspeichern für 2ten Hub ;
 900:  R[45]=(R[4]) ;
 901:  IF (F[98] AND F[732]),R[4]=(R[43]) ;
 902:  !Überprüfungung Zangenstellung ;
 903:  DO[718]=(OFF) ;
 904:  DO[717]=(!DI[717]) ;
 905:  DO[18181]=(ON) ;
 906:  WAIT (DI[717])    ;
 907:  DO[18181]=(OFF) ;
 908:  DO[834]=(ON) ;
 909:  DO[717]=(OFF) ;
 910:  !EZ1/SP1 schliessen ;
 911:  DO[718]=(ON) ;
 912:  !Fraeser ausblasen AUS/EIN ;
 913:  DO[847]=(F[330]) ;
 914:  TIMER[9]=((-4)) ;
 915:  !EZ1/SP1 Kraft erreicht ;
 916:  WAIT ((DI[718] AND !DI[772] AND !DI[780] AND !DI[774] AND !DI[775]) OR (TIMER[9]>=0))    ;
 917:  F[325]=((TIMER[9]>=0)) ;
 918:  DO[18181]=(ON) ;
 919:  DO[718]=((TIMER[9]<0)) ;
 920:  DO[834]=((TIMER[9]<0)) ;
 921:  WAIT ((DI[718] AND !DI[772] AND !DI[780] AND !DI[774] AND !DI[775]) OR DI[26] OR DI[27])    ;
 922:  DO[18181]=(OFF) ;
 923:  !EZ1/SP1 Fehler Kraftaufbau ;
 924:  IF (F[325]),JMP LBL[1201] ;
 925:  TIMER[9]=((-5)) ;
 926:  LBL[1200] ;
 927:  WAIT (!DI[834] OR F[325] OR (TIMER[9]>=0))    ;
 928:  WAIT (DI[834] OR F[325] OR (TIMER[9]>=0))    ;
 929:  R[1]=(R[1]+1) ;
 930:  F[329]=((TIMER[9]>=0)) ;
 931:  !Fraeszeit ueberschritten ;
 932:  IF (F[329]),JMP LBL[1201] ;
 933:  !Umdrehungen Vergleichen ;
 934:  IF (R[1]<R[4]),JMP LBL[1200] ;
 935:  !EZ1/SP1 2 Huebe bei NF ;
 936:  IF (!F[130]),JMP LBL[1201] ;
 937:  IF (F[98]),F[96]=(ON) ;
 938:  F[98]=(ON) ;
 939:  LBL[1201] ;
 940:  DO[834]=((TIMER[9]<0)) ;
 941:  !Fraeser ausblasen EIN ;
 942:  DO[847]=PULSE,4.0sec ;
 943:  !EZ1/SP1 oeffnen ;
 944:  DO[718]=(OFF) ;
 945:  DO[717]=(!DI[717]) ;
 946:  DO[18181]=(F[329]) ;
 947:  WAIT (!F[329] OR DI[26] OR DI[27])    ;
 948:  DO[18181]=(OFF) ;
 949:  DO[18181]=(ON) ;
 950:  WAIT (DI[717])    ;
 951:  DO[18181]=(OFF) ;
 952:  DO[717]=(OFF) ;
 953:  !Umdrehungen ruecksetzen ;
 954:  R[1]=0    ;
 955:  R[42]=12    ;
 956:  !Zähler umschreiben für 2ten Hub ;
 957:  IF (F[98] AND F[732]),GO[3]=36 ;
 958:  IF (F[96] AND F[732]),R[4]=(R[45]) ;
 959:  IF (F[329] OR F[325] OR (!F[96] AND F[130])),JMP LBL[12] ;
 960:  F[98]=(ON) ;
 961:  JMP LBL[13] ;
 962:   ;
 963:  !**************************** ;
 964:  !*        Schritt 13        * ;
 965:  !* STAT EZ1/SP1 i.O./n.i.O. * ;
 966:  !**************************** ;
 967:   ;
 968:  LBL[13] ;
 969:  R[41]=13    ;
 970:  !Fraesueberwachung starten ;
 971:  TIMER[7]=((-5)) ;
 972:  WAIT ((F[78] OR F[79]) AND (F[98] OR (F[94] AND F[96])) OR (TIMER[7]>=0))    ;
 973:  F[329]=((TIMER[7]>=0)) ;
 974:  IF (!F[329]),R[41]=14 ;
 975:  IF (F[329]),R[41]=12 ;
 976:  !KF1 U-Merker ruecksetzen ;
 977:  F[94]=(OFF) ;
 978:  F[96]=(OFF) ;
 979:  F[98]=(OFF) ;
 980:  R[42]=13    ;
 981:  JMP LBL[R[41]] ;
 982:   ;
 983:  !*************************** ;
 984:  !*       Schritt 14        * ;
 985:  !*    STAT EZ1/SP1 KS1     * ;
 986:  !* KS1 in Ruhest.schwenken * ;
 987:  !*************************** ;
 988:   ;
 989:  LBL[14] ;
 990:  R[41]=14    ;
 991:  !RSK gestartet ;
 992:  F[321]=(OFF) ;
 993:  DO[718]=(OFF) ;
 994:  DO[717]=(!DI[717]) ;
 995:  DO[18181]=(ON) ;
 996:  WAIT (DI[717])    ;
 997:  DO[18181]=(OFF) ;
 998:  DO[717]=(OFF) ;
 999:  TIMER[8]=((-4)) ;
1000:  WAIT ((DI[844] AND !DI[842] AND !DI[845] AND DI[843]) OR (TIMER[8]>=0))    ;
1001:  F[324]=((TIMER[8]>=0)) ;
1002:  DO[18181]=((TIMER[8]>=0)) ;
1003:  WAIT (DI[844] AND !DI[842] AND !DI[845] AND DI[843])    ;
1004:  DO[18181]=(OFF) ;
1005:  F[324]=(OFF) ;
1006:  TIMER[8]=((-4)) ;
1007:  DO[835]=(F[564]) ;
1008:  WAIT ((DI[835] AND F[564]) OR (!DI[835] AND !F[564]) OR (TIMER[8]>=0))    ;
1009:  F[323]=((TIMER[8]>=0)) ;
1010:  DO[18181]=((TIMER[8]>=0)) ;
1011:  WAIT ((DI[835] AND F[564]) OR (!DI[835] AND !F[564]))    ;
1012:  DO[18181]=(OFF) ;
1013:  F[323]=(OFF) ;
1014:  !Ueberwachungszeit KS1 Schwenken ;
1015:  TIMER[8]=((-4)) ;
1016:  DO[3969]=(ON) ;
1017:  WAIT (DI[841] OR (TIMER[8]>=0))    ;
1018:  DO[18181]=((TIMER[8]>=0)) ;
1019:  WAIT (DI[841])    ;
1020:  DO[18181]=(OFF) ;
1021:  TIMER[8]=((-6)) ;
1022:  WAIT ((!DI[844] AND DI[842] AND DI[845] AND !DI[843]) OR (TIMER[8]>=0))    ;
1023:  F[323]=((TIMER[8]>=0)) ;
1024:  DO[3969]=(OFF) ;
1025:  DO[18181]=((TIMER[8]>=0)) ;
1026:  WAIT ((!DI[844] AND DI[842] AND DI[845] AND !DI[843]) OR DI[26])    ;
1027:  DO[18181]=(OFF) ;
1028:  DO[835]=(OFF) ;
1029:  F[323]=(OFF) ;
1030:  DO[834]=(OFF) ;
1031:  !Sprung zurueck bei KS1 Fehler ;
1032:  IF (TIMER[8]>=0),JMP LBL[14] ;
1033:  R[42]=14    ;
1034:  JMP LBL[15] ;
1035:   ;
1036:  !*********************** ;
1037:  !*     Schritt 15      * ;
1038:  !*    STAT EZ1/SP1     * ;
1039:  !*  STAT EZ1/SP1/KE1   * ;
1040:  !* Messen nach Fraesen * ;
1041:  !*********************** ;
1042:   ;
1043:  LBL[15] ;
1044:  R[41]=15    ;
1045:  !RSK gestartet ;
1046:  F[321]=(OFF) ;
1047:  GO[3]=1 ;
1048:  WAIT    .10(sec) ;
1049:  DO[786]=(!F[830]) ;
1050:  DO[722]=(F[830]) ;
1051:  DO[18181]=(ON) ;
1052:  WAIT ((!DI[786] AND DI[787] AND !DI[788]) OR F[830])    ;
1053:  WAIT ((!DI[722] AND DI[724] AND !DI[723] OR F[329]) OR !F[830])    ;
1054:  DO[18181]=(OFF) ;
1055:  DO[786]=(F[830] AND DO[786]) ;
1056:  DO[722]=(!F[830] AND DO[722]) ;
1057:  GO[1]=(31) ;
1058:  GO[3]=(31) ;
1059:  WAIT    .10(sec) ;
1060:  DO[757]=(ON) ;
1061:  TIMER[9]=((-8)) ;
1062:  WAIT (DI[757] OR (TIMER[9]>=0))    ;
1063:  F[326]=((TIMER[9]>=0)) ;
1064:  DO[18181]=(ON) ;
1065:  WAIT (DI[757] OR DI[26] OR DI[27])    ;
1066:  DO[18181]=(OFF) ;
1067:  F[326]=(OFF) ;
1068:  F[85]=(DI[776] OR DI[777]) ;
1069:  DO[757]=(OFF) ;
1070:  F[86]=(DI[736] OR (DI[735] AND DI[734] AND DI[733])) ;
1071:  TIMER[7]=((-2)) ;
1072:  WAIT ((!F[85] AND !F[86]) OR (TIMER[7]>=0))    ;
1073:  F[329]=((TIMER[7]>=0)) ;
1074:  DO[18181]=(F[329]) ;
1075:  WAIT ((!F[85] AND !F[86]) OR DI[26] OR DI[27])    ;
1076:  DO[18181]=(OFF) ;
1077:  F[329]=(OFF) ;
1078:  F[298]=(F[85] OR F[86]) ;
1079:  DO[717]=(!DI[717]) ;
1080:  DO[18181]=(ON) ;
1081:  WAIT ((DI[717] AND !DI[784]) OR (DI[717] AND F[298]))    ;
1082:  DO[18181]=(OFF) ;
1083:  DO[717]=(OFF) ;
1084:  R[42]=15    ;
1085:  !EZ1/SP1 wiederh. bei Messfehler ;
1086:  IF (DI[777]),JMP LBL[17] ;
1087:  DO[758]=(OFF) ;
1088:  DO[759]=(OFF) ;
1089:  !KS nicht bei K-Verschleiss ;
1090:  IF (F[298]),JMP LBL[9] ;
1091:  !EZ1/SP1 2.Setzhub nach Fraesen ;
1092:  IF (F[335] AND F[78]),JMP LBL[55] ;
1093:  !EZ1/SP1 Kurzschluss schweissen ;
1094:  IF (F[335] AND !F[78]),JMP LBL[16] ;
1095:  !EZ1/SP1 Kurzschluss schweissen ;
1096:  IF (!F[335]),JMP LBL[16] ;
1097:   ;
1098:  !************************** ;
1099:  !*       Schritt 16       * ;
1100:  !*      STAT EZ1/SP1      * ;
1101:  !* Kurzschlussschweissung * ;
1102:  !************************** ;
1103:   ;
1104:  LBL[16] ;
1105:  R[41]=16    ;
1106:  !RSK gestartet ;
1107:  F[321]=(OFF) ;
1108:  DO[145]=(ON) ;
1109:  !EZ1/SK1 Prog. ;
1110:  IF (F[78] AND !F[301]),GO[1]=(41) ;
1111:  IF (F[78] AND !F[301]),GO[3]=(41) ;
1112:  IF (F[79] OR F[301]),GO[1]=(51) ;
1113:  IF (F[79] OR F[301]),GO[3]=(51) ;
1114:  WAIT    .10(sec) ;
1115:  DO[717]=(OFF) ;
1116:  DO[718]=(OFF) ;
1117:  DO[785]=(OFF) ;
1118:  DO[514]=(OFF) ;
1119:  F[80]=(OFF) ;
1120:  F[306]=(OFF) ;
1121:  DO[18181]=(ON) ;
1122:  WAIT (DI[705] AND DI[713] AND DI[714] AND (!DI[784] OR (DI[769] AND DI[784])))    ;
1123:  DO[18181]=(OFF) ;
1124:  F[346]=(OFF) ;
1125:  DO[18181]=(ON) ;
1126:  WAIT ((!DI[785] AND DI[792] AND DI[802] AND !F[80]) OR (!DI[792] AND DI[802] AND DI[145]))    ;
1127:  DO[18181]=(OFF) ;
1128:  !EZ1/SP1 schliessen ;
1129:  DO[718]=(ON) ;
1130:  TIMER[9]=((-4)) ;
1131:  !EZ1/SP1 Kraft erreicht ;
1132:  WAIT ((DI[718] AND !DI[772] AND !DI[780]) OR DI[774] OR DI[775] OR (TIMER[9]>=0))    ;
1133:  DO[718]=(DI[718] AND !DI[774] AND !DI[775]) ;
1134:  DO[717]=(!DO[718]) ;
1135:  !Schweissen START ;
1136:  DO[785]=(DI[718] AND !DI[774] AND !DI[775]) ;
1137:  !EZ1/SP1 Fehler Ausgleich ;
1138:  F[302]=(DI[718] AND DI[719]) ;
1139:  !EZ1/SP1 Fehler SZ ;
1140:  F[300]=(DI[774] OR DI[775]) ;
1141:  !SK1 FK ;
1142:  TIMER[9]=((-1)) ;
1143:  WAIT ((F[80] AND DO[785]) OR ((DI[804] OR DI[805]) AND (DI[785] AND DO[785])) OR (DI[771] AND DI[784]) OR !DO[785] OR (TIMER[9]>=0))    ;
1144:  F[297]=(F[80] OR (DI[804] AND !DI[806] AND !DI[775] AND DI[785])) ;
1145:  !Fehler SK1 ;
1146:  F[301]=(!F[297] AND !F[298] AND DO[785]) ;
1147:  DO[785]=(OFF) ;
1148:  DO[718]=(OFF) ;
1149:  DO[18181]=(ON) ;
1150:  F[749]=(!F[297] AND !F[748]) ;
1151:  F[748]=(!F[297]) ;
1152:  WAIT (F[297] OR DI[26] OR DI[27] OR (F[749] AND F[731]))    ;
1153:  DO[910]=(OFF) ;
1154:  WAIT (!DI[26] AND !DI[27])    ;
1155:  DO[18181]=(OFF) ;
1156:  !EZ1/SP1 oeffnen ;
1157:  DO[717]=(!DI[717]) ;
1158:  TIMER[9]=((-4)) ;
1159:  WAIT (DI[717] OR (TIMER[9]>=0))    ;
1160:  F[303]=((TIMER[9]>=0)) ;
1161:  DO[18181]=(F[303]) ;
1162:  WAIT (DI[717])    ;
1163:  DO[18181]=(OFF) ;
1164:  F[303]=(OFF) ;
1165:  DO[717]=(OFF) ;
1166:  DO[145]=(OFF) ;
1167:  R[42]=16    ;
1168:  JMP LBL[17] ;
1169:   ;
1170:  !************************** ;
1171:  !*       Schritt 17       * ;
1172:  !*      STAT EZ1/SP1      * ;
1173:  !************************** ;
1174:   ;
1175:  LBL[17] ;
1176:  R[41]=17    ;
1177:  !RSK gestartet ;
1178:  F[321]=(OFF) ;
1179:  !Sprung zurueck bei Fehler ;
1180:  IF (!F[297] AND !DI[777]),JMP LBL[9] ;
1181:  !STAT EZ1/SP1 FK Fraesen ;
1182:  F[93]=(!F[329]) ;
1183:  DO[116]=(OFF) ;
1184:  DO[130]=(OFF) ;
1185:  R[42]=17    ;
1186:  JMP LBL[1] ;
1187:   ;
1188:   ;
1189:  !************************ ;
1190:  !************************ ;
1191:  !* Fraesen STAT EZ2/SP2 * ;
1192:  !************************ ;
1193:  !************************ ;
1194:   ;
1195:   ;
1196:  !****************************** ;
1197:  !*        Schritt 18          * ;
1198:  !*     STAT EZ2/SP2 KS2       * ;
1199:  !* KS2 in Arbeitsst.schwenken * ;
1200:  !****************************** ;
1201:   ;
1202:  LBL[18] ;
1203:  R[41]=18    ;
1204:  !RSK gestartet ;
1205:  F[321]=(OFF) ;
1206:  GO[4]=(31) ;
1207:  IF (F[285]),GO[3]=(35) ;
1208:  IF (!F[285]),GO[6]=(31) ;
1209:  WAIT    .10(sec) ;
1210:  DO[918]=(F[138]) ;
1211:  DO[919]=(F[139]) ;
1212:  DO[116]=(ON) ;
1213:  DO[162]=(ON) ;
1214:  DO[878]=(OFF) ;
1215:  DO[877]=(!DI[877]) ;
1216:  DO[18181]=(ON) ;
1217:  WAIT (DI[877])    ;
1218:  DO[18181]=(OFF) ;
1219:  DO[877]=(OFF) ;
1220:  !Ueberwachungszeit Grundstellung ;
1221:  TIMER[8]=((-4)) ;
1222:  WAIT ((!DI[1004] AND DI[1002] AND DI[1005] AND !DI[1003]) OR (TIMER[8]>=0))    ;
1223:  F[323]=((TIMER[8]>=0)) ;
1224:  DO[18181]=((TIMER[8]>=0)) ;
1225:  WAIT (!DI[1004] AND DI[1002] AND DI[1005] AND !DI[1003])    ;
1226:  DO[18181]=(OFF) ;
1227:  F[323]=(OFF) ;
1228:  TIMER[8]=((-4)) ;
1229:  DO[995]=(F[564]) ;
1230:  WAIT ((DI[995] AND F[564]) OR (!DI[995] AND !F[564]) OR (TIMER[8]>=0))    ;
1231:  F[323]=((TIMER[8]>=0)) ;
1232:  DO[18181]=((TIMER[8]>=0)) ;
1233:  WAIT ((DI[995] AND F[564]) OR (!DI[995] AND !F[564]))    ;
1234:  DO[18181]=(OFF) ;
1235:  F[323]=(OFF) ;
1236:  !Ueberwachungszeit KS2 Schwenken ;
1237:  TIMER[8]=((-6)) ;
1238:  DO[3973]=(ON) ;
1239:  DO[18181]=(ON) ;
1240:  WAIT (DI[1001])    ;
1241:  DO[18181]=(OFF) ;
1242:  WAIT ((DI[1004] AND !DI[1002] AND !DI[1005] AND DI[1003]) OR (TIMER[8]>=0))    ;
1243:  F[324]=((TIMER[8]>=0)) ;
1244:  DO[3973]=(OFF) ;
1245:  DO[18181]=((TIMER[8]>=0)) ;
1246:  WAIT ((DI[1004] AND !DI[1002] AND !DI[1005] AND DI[1003]) OR DI[26])    ;
1247:  DO[18181]=(OFF) ;
1248:  F[324]=(OFF) ;
1249:  !Sprung zurueck bei KS2 Fehler ;
1250:  IF (TIMER[8]>=0),JMP LBL[18] ;
1251:  DO[995]=(OFF) ;
1252:  TIMER[11]=((R[24])) ;
1253:  WAIT ((TIMER[11]>=0) OR !F[564])    ;
1254:  TIMER[11]=STOP ;
1255:  DO[18181]=(ON) ;
1256:  WAIT ((F[148] AND F[138]) OR (F[148] AND F[139]))    ;
1257:  DO[18181]=(OFF) ;
1258:  !Anwahl Startfraesen ;
1259:  IF (!DI[1002] AND DI[1003] AND F[148] AND F[138] AND !F[301]),R[41]=19 ;
1260:  !Anwahl Normalfraesen ;
1261:  IF (!DI[1002] AND DI[1003] AND F[148] AND (F[139] OR F[301])),R[41]=21 ;
1262:  R[42]=18    ;
1263:  JMP LBL[R[41]] ;
1264:   ;
1265:  !************************** ;
1266:  !*      Schritt 19        * ;
1267:  !* STAT EZ2/SP2 SF Teil 1 * ;
1268:  !************************** ;
1269:   ;
1270:  LBL[19] ;
1271:  R[41]=19    ;
1272:  !RSK gestartet ;
1273:  F[321]=(OFF) ;
1274:  F[329]=(OFF) ;
1275:  F[325]=(OFF) ;
1276:  DO[878]=(OFF) ;
1277:  DO[877]=(!DI[877]) ;
1278:  DO[18181]=(ON) ;
1279:  WAIT (DI[877])    ;
1280:  DO[18181]=(OFF) ;
1281:  DO[994]=(ON) ;
1282:  DO[877]=(OFF) ;
1283:  !Warte Fraeser laeuft ;
1284:  TIMER[7]=((-3)) ;
1285:  WAIT (!DI[994] OR (TIMER[7]>=0))    ;
1286:  WAIT (DI[994] OR (TIMER[7]>=0))    ;
1287:  F[322]=((TIMER[7]>=0)) ;
1288:  DO[18181]=(ON) ;
1289:  WAIT (!DI[994])    ;
1290:  WAIT (DI[994])    ;
1291:  DO[18181]=(OFF) ;
1292:  F[322]=(OFF) ;
1293:  !EZ2/SP2 schliessen ;
1294:  DO[878]=(ON) ;
1295:  !Fraeser ausblasen AUS/EIN ;
1296:  DO[1007]=(F[330]) ;
1297:  TIMER[9]=((-4)) ;
1298:  !EZ2/SP2 Kraft erreicht ;
1299:  WAIT ((DI[878] AND !DI[932] AND !DI[940] AND !DI[934] AND !DI[935]) OR (TIMER[9]>=0))    ;
1300:  F[325]=((TIMER[9]>=0)) ;
1301:  DO[18181]=(ON) ;
1302:  DO[878]=((TIMER[9]<0)) ;
1303:  DO[994]=((TIMER[9]<0)) ;
1304:  WAIT ((DI[878] AND !DI[932] AND !DI[940] AND !DI[934] AND !DI[935]) OR DI[26] OR DI[27])    ;
1305:  DO[18181]=(OFF) ;
1306:  F[325]=(OFF) ;
1307:  !EZ2/SP2 Fehler Kraftaufbau ;
1308:  IF (F[325]),JMP LBL[1901] ;
1309:  TIMER[9]=((-5)) ;
1310:  LBL[1900] ;
1311:  WAIT (!DI[994] OR F[325] OR (TIMER[9]>=0))    ;
1312:  WAIT (DI[994] OR F[325] OR (TIMER[9]>=0))    ;
1313:  R[1]=(R[1]+1) ;
1314:  F[329]=((TIMER[9]>=0)) ;
1315:  !Fraeszeit ueberschritten ;
1316:  IF (F[329]),JMP LBL[1901] ;
1317:  !Umdrehungen Vergleichen ;
1318:  IF (R[1]<R[5]),JMP LBL[1900] ;
1319:  F[150]=(ON) ;
1320:  LBL[1901] ;
1321:  DO[994]=((TIMER[9]<0)) ;
1322:  !Fraeser ausblasen EIN ;
1323:  DO[1007]=(F[330] OR (TIMER[9]<0)) ;
1324:  DO[878]=(OFF) ;
1325:  !EZ2/SP2 oeffnen ;
1326:  DO[877]=(!DI[877]) ;
1327:  DO[18181]=(F[329]) ;
1328:  WAIT (!F[329] OR DI[26] OR DI[27])    ;
1329:  DO[18181]=(OFF) ;
1330:  DO[18181]=(ON) ;
1331:  WAIT (DI[877])    ;
1332:  DO[18181]=(OFF) ;
1333:  DO[877]=(OFF) ;
1334:  !Umdrehungen ruecksetzen ;
1335:  R[1]=0    ;
1336:  R[42]=19    ;
1337:  IF (F[329] OR F[325]),JMP LBL[19] ;
1338:  JMP LBL[20] ;
1339:   ;
1340:  !************************** ;
1341:  !*       Schritt 20       * ;
1342:  !* STAT EZ2/SP2 SF Teil 2 * ;
1343:  !************************** ;
1344:   ;
1345:  LBL[20] ;
1346:  R[41]=20    ;
1347:  !RSK gestartet ;
1348:  F[321]=(OFF) ;
1349:  F[329]=(OFF) ;
1350:  F[325]=(OFF) ;
1351:  DO[878]=(OFF) ;
1352:  DO[877]=(!DI[877]) ;
1353:  DO[18181]=(ON) ;
1354:  WAIT (DI[877])    ;
1355:  DO[18181]=(OFF) ;
1356:  DO[994]=(ON) ;
1357:  DO[877]=(OFF) ;
1358:  !Zange zu... ;
1359:  DO[878]=(ON) ;
1360:  !Fraeser ausblasen AUS/EIN ;
1361:  DO[1007]=(F[330]) ;
1362:  TIMER[9]=((-4)) ;
1363:  !EZ2/SP2 Kraft erreicht ;
1364:  WAIT ((DI[878] AND !DI[932] AND !DI[940] AND !DI[934] AND !DI[935]) OR (TIMER[9]>=0))    ;
1365:  F[325]=((TIMER[9]>=0)) ;
1366:  DO[18181]=(ON) ;
1367:  DO[878]=((TIMER[9]<0)) ;
1368:  DO[994]=((TIMER[9]<0)) ;
1369:  WAIT ((DI[878] AND !DI[932] AND !DI[940] AND !DI[934] AND !DI[935]) OR DI[26] OR DI[27])    ;
1370:  DO[18181]=(OFF) ;
1371:  !EZ2/SP2 Fehler Kraftaufbau ;
1372:  IF (F[325]),JMP LBL[2001] ;
1373:  TIMER[9]=((-5)) ;
1374:  LBL[2000] ;
1375:  WAIT (!DI[994] OR F[325] OR (TIMER[9]>=0))    ;
1376:  WAIT (DI[994] OR F[325] OR (TIMER[9]>=0))    ;
1377:  R[1]=(R[1]+1) ;
1378:  F[329]=((TIMER[9]>=0)) ;
1379:  !Fraeszeit ueberschritten ;
1380:  IF (F[329]),JMP LBL[2001] ;
1381:  !Umdrehungen Vergleichen ;
1382:  IF (R[1]<R[6]),JMP LBL[2000] ;
1383:  F[152]=(ON) ;
1384:  LBL[2001] ;
1385:  DO[994]=((TIMER[9]<0)) ;
1386:  !Fraeser ausblasen EIN ;
1387:  DO[1007]=PULSE,4.0sec ;
1388:  DO[878]=(OFF) ;
1389:  !EZ2/SP2 oeffnen ;
1390:  DO[877]=(!DI[877]) ;
1391:  DO[18181]=(F[329]) ;
1392:  WAIT (!F[329] OR DI[26] OR DI[27])    ;
1393:  DO[18181]=(OFF) ;
1394:  DO[18181]=(ON) ;
1395:  WAIT (DI[877])    ;
1396:  DO[18181]=(OFF) ;
1397:  DO[877]=(OFF) ;
1398:  !Umdrehungen ruecksetzen ;
1399:  R[1]=0    ;
1400:  R[42]=20    ;
1401:  IF (F[329] OR F[325]),JMP LBL[20] ;
1402:  JMP LBL[22] ;
1403:   ;
1404:  !********************* ;
1405:  !*     Schritt 21    * ;
1406:  !*   STAT EZ2/SP2 NF * ;
1407:  !********************* ;
1408:   ;
1409:  LBL[21] ;
1410:  R[41]=21    ;
1411:  !RSK gestartet ;
1412:  F[321]=(OFF) ;
1413:  F[329]=(OFF) ;
1414:  F[325]=(OFF) ;
1415:  !Zähler wegspeichern für 2ten Hub ;
1416:  R[45]=(R[7]) ;
1417:  IF (F[154] AND F[732]),R[7]=(R[44]) ;
1418:  DO[878]=(OFF) ;
1419:  DO[877]=(!DI[877]) ;
1420:  DO[18181]=(ON) ;
1421:  WAIT (DI[877])    ;
1422:  DO[18181]=(OFF) ;
1423:  DO[994]=(ON) ;
1424:  DO[877]=(OFF) ;
1425:  !EZ2/SP2 schliessen ;
1426:  DO[878]=(ON) ;
1427:  !Fraeser ausblasen AUS ;
1428:  DO[1007]=(F[330]) ;
1429:  TIMER[9]=((-4)) ;
1430:  !EZ2/SP2 Kraft erreicht ;
1431:  WAIT ((DI[878] AND !DI[932] AND !DI[940] AND !DI[934] AND !DI[935]) OR (TIMER[9]>=0))    ;
1432:  F[325]=((TIMER[9]>=0)) ;
1433:  DO[18181]=(ON) ;
1434:  DO[878]=((TIMER[9]<0)) ;
1435:  DO[994]=((TIMER[9]<0)) ;
1436:  WAIT ((DI[878] AND !DI[932] AND !DI[940] AND !DI[934] AND !DI[935]) OR DI[26] OR DI[27])    ;
1437:  DO[18181]=(OFF) ;
1438:  !EZ2/SP2 Fehler Kraftaufbau ;
1439:  IF (F[325]),JMP LBL[2101] ;
1440:  TIMER[9]=((-5)) ;
1441:  LBL[2100] ;
1442:  WAIT (!DI[994] OR F[325] OR (TIMER[9]>=0))    ;
1443:  WAIT (DI[994] OR F[325] OR (TIMER[9]>=0))    ;
1444:  R[1]=(R[1]+1) ;
1445:  F[329]=((TIMER[9]>=0)) ;
1446:  !Fraeszeit ueberschritten ;
1447:  IF (F[329]),JMP LBL[2101] ;
1448:  !Umdrehungen Vergleichen ;
1449:  IF (R[1]<R[7]),JMP LBL[2100] ;
1450:  !EZ2/SP2 2 Huebe bei NF ;
1451:  IF (!F[164]),JMP LBL[2101] ;
1452:  IF (F[154]),F[152]=(ON) ;
1453:  F[154]=(ON) ;
1454:  LBL[2101] ;
1455:  DO[878]=(OFF) ;
1456:  DO[994]=((TIMER[9]<0)) ;
1457:  !Fraeser ausblasen EIN ;
1458:  DO[1007]=PULSE,4.0sec ;
1459:  !EZ2/SP2 oeffnen ;
1460:  DO[877]=(!DI[877]) ;
1461:  DO[18181]=(F[329]) ;
1462:  WAIT (!F[329] OR DI[26] OR DI[27])    ;
1463:  DO[18181]=(OFF) ;
1464:  DO[18181]=(ON) ;
1465:  WAIT (DI[877])    ;
1466:  DO[18181]=(OFF) ;
1467:  DO[877]=(OFF) ;
1468:  !Umdrehungen ruecksetzen ;
1469:  R[1]=0    ;
1470:  R[42]=21    ;
1471:  !Zähler umschreiben für 2ten Hub ;
1472:  IF (F[154] AND F[732]),GO[3]=36 ;
1473:  IF (F[152] AND F[732]),R[7]=(R[45]) ;
1474:  IF (F[329] OR F[325] OR (!F[152] AND F[164])),JMP LBL[21] ;
1475:  F[154]=(ON) ;
1476:  JMP LBL[22] ;
1477:   ;
1478:  !*************************** ;
1479:  !*        Schritt 22       * ;
1480:  !* STAT EZ2/SP2 i.O/n.i.O. * ;
1481:  !*************************** ;
1482:   ;
1483:  LBL[22] ;
1484:  R[41]=22    ;
1485:  !Fraesueberwachung starten ;
1486:  TIMER[7]=((-5)) ;
1487:  WAIT ((F[138] OR F[139]) AND (F[154] OR (F[150] AND F[152])) OR (TIMER[7]>=0))    ;
1488:  F[329]=((TIMER[7]>=0)) ;
1489:  IF (!F[329]),R[41]=23 ;
1490:  IF (F[329]),R[41]=21 ;
1491:  !KF1 U-Merker ruecksetzen ;
1492:  F[150]=(OFF) ;
1493:  F[152]=(OFF) ;
1494:  F[154]=(OFF) ;
1495:  R[42]=22    ;
1496:  JMP LBL[R[41]] ;
1497:   ;
1498:  !*************************** ;
1499:  !*       Schritt 23        * ;
1500:  !*      STAT EZ2/SP2       * ;
1501:  !* KS2 in Ruhest.schwenken * ;
1502:  !*************************** ;
1503:   ;
1504:  LBL[23] ;
1505:  R[41]=23    ;
1506:  !RSK gestartet ;
1507:  F[321]=(OFF) ;
1508:  DO[878]=(OFF) ;
1509:  DO[877]=(!DI[877]) ;
1510:  DO[18181]=(ON) ;
1511:  WAIT (DI[877])    ;
1512:  DO[18181]=(OFF) ;
1513:  DO[877]=(OFF) ;
1514:  TIMER[8]=((-4)) ;
1515:  WAIT ((DI[1004] AND !DI[1002] AND !DI[1005] AND DI[1003]) OR (TIMER[8]>=0))    ;
1516:  F[324]=((TIMER[8]>=0)) ;
1517:  DO[18181]=((TIMER[8]>=0)) ;
1518:  WAIT (DI[1004] AND !DI[1002] AND !DI[1005] AND DI[1003])    ;
1519:  DO[18181]=(OFF) ;
1520:  F[324]=(OFF) ;
1521:  TIMER[8]=((-4)) ;
1522:  DO[995]=(F[564]) ;
1523:  WAIT ((DI[995] AND F[564]) OR (!DI[995] AND !F[564]) OR (TIMER[8]>=0))    ;
1524:  F[323]=((TIMER[8]>=0)) ;
1525:  DO[18181]=((TIMER[8]>=0)) ;
1526:  WAIT ((DI[995] AND F[564]) OR (!DI[995] AND !F[564]))    ;
1527:  DO[18181]=(OFF) ;
1528:  F[323]=(OFF) ;
1529:  !Ueberwachungszeit KS2 Schwenken ;
1530:  TIMER[8]=((-4)) ;
1531:  DO[3970]=(ON) ;
1532:  WAIT (DI[1001] OR (TIMER[8]>=0))    ;
1533:  DO[18181]=((TIMER[8]>=0)) ;
1534:  WAIT (DI[1001])    ;
1535:  TIMER[8]=((-6)) ;
1536:  DO[18181]=(OFF) ;
1537:  WAIT ((!DI[1004] AND DI[1002] AND DI[1005] AND !DI[1003]) OR (TIMER[8]>=0))    ;
1538:  F[323]=((TIMER[8]>=0)) ;
1539:  DO[3970]=(OFF) ;
1540:  DO[18181]=((TIMER[8]>=0)) ;
1541:  WAIT ((!DI[1004] AND DI[1002] AND DI[1005] AND !DI[1003]) OR DI[26])    ;
1542:  DO[18181]=(OFF) ;
1543:  F[323]=(OFF) ;
1544:  DO[995]=(OFF) ;
1545:  DO[994]=(OFF) ;
1546:  !Sprung zurueck bei KS2 Fehler ;
1547:  IF (TIMER[8]>=0),JMP LBL[23] ;
1548:  R[42]=23    ;
1549:  JMP LBL[24] ;
1550:   ;
1551:  !*********************** ;
1552:  !*     Schritt 24      * ;
1553:  !*    STAT EZ2/SP2     * ;
1554:  !* Messen nach Fraesen * ;
1555:  !*********************** ;
1556:   ;
1557:  LBL[24] ;
1558:  R[41]=24    ;
1559:  !RSK gestartet ;
1560:  F[321]=(OFF) ;
1561:  IF (!F[285]),JMP LBL[2400] ;
1562:  IF (F[285]),JMP LBL[2401] ;
1563:  LBL[2400] ;
1564:  GO[6]=1 ;
1565:  WAIT    .10(sec) ;
1566:  DO[946]=(!F[831]) ;
1567:  DO[882]=(F[831]) ;
1568:  !STAT EZ2/SP2 FK Fraesen ;
1569:  DO[18181]=(ON) ;
1570:  WAIT ((!DI[946] AND DI[947] AND !DI[948]) OR F[831])    ;
1571:  WAIT ((!DI[882] AND DI[883]) OR !F[831])    ;
1572:  DO[18181]=(OFF) ;
1573:  DO[946]=(F[831]) ;
1574:  DO[882]=(!F[831]) ;
1575:  JMP LBL[2402] ;
1576:  LBL[2401] ;
1577:  IF (!F[285]),GO[3]=(1) ;
1578:  IF (F[285]),GO[3]=(5) ;
1579:  WAIT    .10(sec) ;
1580:  DO[786]=(ON) ;
1581:  !STAT EZ2/SP2 FK Fraesen ;
1582:  DO[18181]=(ON) ;
1583:  WAIT (!DI[786] AND DI[787] AND !DI[788])    ;
1584:  DO[18181]=(OFF) ;
1585:  DO[786]=(OFF) ;
1586:  LBL[2402] ;
1587:  GO[4]=(31) ;
1588:  IF (F[285]),GO[3]=(35) ;
1589:  IF (!F[285]),GO[6]=(31) ;
1590:  WAIT    .10(sec) ;
1591:  DO[917]=(ON) ;
1592:  TIMER[9]=((-8)) ;
1593:  WAIT (DI[917] OR (TIMER[9]>=0))    ;
1594:  F[326]=((TIMER[9]>=0)) ;
1595:  DO[18181]=(F[326]) ;
1596:  WAIT (DI[917] OR DI[26] OR DI[27])    ;
1597:  DO[18181]=(OFF) ;
1598:  F[326]=(OFF) ;
1599:  F[143]=(DI[936] OR DI[937]) ;
1600:  DO[917]=(OFF) ;
1601:  F[144]=(DI[896] OR (DI[895] AND DI[894] AND DI[893])) ;
1602:  TIMER[7]=((-2)) ;
1603:  WAIT ((!F[144] AND !F[143]) OR (TIMER[7]>=0))    ;
1604:  F[329]=((TIMER[7]>=0)) ;
1605:  DO[18181]=(F[329]) ;
1606:  WAIT ((!F[144] AND !F[143]) OR DI[26] OR DI[27])    ;
1607:  DO[18181]=(OFF) ;
1608:  F[329]=(OFF) ;
1609:  F[298]=(F[144] OR F[143]) ;
1610:  DO[877]=(!DI[877]) ;
1611:  DO[18181]=(ON) ;
1612:  WAIT ((DI[877] AND !DI[944]) OR (DI[877] AND F[298]))    ;
1613:  DO[18181]=(OFF) ;
1614:  DO[877]=(OFF) ;
1615:  R[42]=24    ;
1616:  !EZ2/SP2 wiederh. bei Messfehler ;
1617:  IF (F[298]),JMP LBL[18] ;
1618:  DO[918]=(OFF) ;
1619:  DO[919]=(OFF) ;
1620:  !KS nicht bei K-Verschleiss ;
1621:  IF (DI[937]),JMP LBL[26] ;
1622:  !EZ2/SP2 2.Setzhub nach Fraesen ;
1623:  IF (F[335] AND F[138]),JMP LBL[56] ;
1624:  !EZ2/SP2 Kurzschluss schweissen ;
1625:  IF (F[335] AND !F[138]),JMP LBL[25] ;
1626:  !EZ2/SP2 Kurzschluss schweissen ;
1627:  IF (!F[335]),JMP LBL[25] ;
1628:   ;
1629:  !************************** ;
1630:  !*       Schritt 25       * ;
1631:  !*      STAT EZ2/SP2      * ;
1632:  !* Kurzschlussschweissung * ;
1633:  !************************** ;
1634:   ;
1635:  LBL[25] ;
1636:  R[41]=25    ;
1637:  !RSK gestartet ;
1638:  F[321]=(OFF) ;
1639:  DO[145]=(F[285]) ;
1640:  DO[177]=(!F[285]) ;
1641:  !EZ2/SP2 SK1/SK2 Prog. ;
1642:  IF (F[285] AND F[138] AND !F[301]),GO[3]=(45) ;
1643:  IF (!F[285] AND F[138] AND !F[301]),GO[4]=(41) ;
1644:  IF (!F[285] AND F[138] AND !F[301]),GO[6]=(41) ;
1645:  IF ((F[285] AND F[139]) OR (F[285] AND F[301])),GO[3]=(55) ;
1646:  IF ((!F[285] AND F[139]) OR (!F[285] AND F[301])),GO[4]=(51) ;
1647:  IF ((!F[285] AND F[139]) OR (!F[285] AND F[301])),GO[6]=(51) ;
1648:  WAIT    .10(sec) ;
1649:  DO[877]=(OFF) ;
1650:  DO[878]=(OFF) ;
1651:  DO[945]=(OFF) ;
1652:  DO[785]=(!F[285] AND DO[785]) ;
1653:  DO[514]=(ON) ;
1654:  F[140]=(OFF) ;
1655:  F[80]=(OFF) ;
1656:  F[142]=(!F[285]) ;
1657:  F[306]=(OFF) ;
1658:  F[303]=(!DI[929] AND DI[944]) ;
1659:  DO[18181]=(ON) ;
1660:  WAIT (DI[865] AND DI[873] AND DI[874] AND (!DI[944] OR (DI[929] AND DI[944])))    ;
1661:  F[303]=(OFF) ;
1662:  WAIT ((!DI[945] AND DI[952] AND DI[962] AND !F[140]) OR (!DI[952] AND DI[962] AND !DI[913]) OR F[285])    ;
1663:  WAIT ((!DI[785] AND DI[792] AND DI[802] AND !F[80]) OR (!DI[792] AND DI[802] AND !DI[913]) OR !F[285])    ;
1664:  DO[18181]=(OFF) ;
1665:  !EZ2/SP2 schliessen ;
1666:  DO[878]=(ON) ;
1667:  TIMER[9]=((-4)) ;
1668:  WAIT ((DI[878] AND !DI[932] AND !DI[940]) OR DI[934] OR DI[935] OR (TIMER[9]>=0))    ;
1669:  DO[878]=(DI[878] AND !DI[934] AND !DI[935]) ;
1670:  DO[877]=(!DO[878]) ;
1671:  !Schweissen START ;
1672:  DO[945]=(DI[878] AND !DI[934] AND !DI[935] AND !F[285]) ;
1673:  DO[785]=((DI[878] AND !DI[934] AND !DI[935] AND F[285]) OR (!F[285] AND DO[785])) ;
1674:  !EZ2/SP2 Fehler Ausgleich ;
1675:  F[302]=(DI[878] AND DI[879]) ;
1676:  !EZ2/SP2 Fehler SZ ;
1677:  F[300]=(DI[934] OR DI[935]) ;
1678:  !SK1/SK2 FK ;
1679:  TIMER[9]=((-10)) ;
1680:  WAIT ((F[140] AND DO[945]) OR ((DI[964] OR DI[965]) AND (DI[945] AND DO[945])) OR (DI[931] AND DI[944]) OR (!DO[945] AND F[285]) OR (TIMER[9]>=0))    ;
1681:  WAIT ((F[80] AND DO[785]) OR ((DI[804] OR DI[805]) AND (DI[785] AND DO[785])) OR (DI[931] AND DI[944]) OR (!DO[785] AND !F[285]) OR (TIMER[9]>=0))    ;
1682:  F[297]=(F[140] OR (!DI[935] AND DI[945] AND DI[964] AND !DI[966]) OR F[80] OR (!DI[935] AND DI[785] AND DI[804] AND !DI[806])) ;
1683:  !Fehler SK1/SK2 ;
1684:  F[301]=(!F[297] AND !F[298] AND (DO[785] OR DO[945])) ;
1685:  DO[945]=(OFF) ;
1686:  DO[878]=(OFF) ;
1687:  DO[785]=((F[285] AND !DI[785]) OR (!F[285] AND DO[785])) ;
1688:  F[327]=(!F[297]) ;
1689:  DO[18181]=(F[327]) ;
1690:  F[749]=(!F[297] AND !F[748]) ;
1691:  F[748]=(!F[297]) ;
1692:  WAIT (F[297] OR DI[26] OR DI[27] OR (F[749] AND F[731]))    ;
1693:  F[327]=(OFF) ;
1694:  WAIT (!DI[26] AND !DI[27])    ;
1695:  DO[18181]=(OFF) ;
1696:  !EZ2/SP2 oeffnen ;
1697:  DO[877]=(!DI[877]) ;
1698:  TIMER[9]=((-4)) ;
1699:  WAIT (DI[877] OR (TIMER[9]>=0))    ;
1700:  F[303]=((TIMER[9]>=0)) ;
1701:  DO[18181]=(F[303]) ;
1702:  WAIT (DI[877])    ;
1703:  DO[18181]=(OFF) ;
1704:  F[303]=(OFF) ;
1705:  DO[877]=(OFF) ;
1706:  DO[145]=(OFF) ;
1707:  DO[177]=(OFF) ;
1708:  R[42]=25    ;
1709:  JMP LBL[26] ;
1710:   ;
1711:  !****************************** ;
1712:  !*         Schritt 26         * ;
1713:  !*       STAT EZ2/SP2 FK      * ;
1714:  !****************************** ;
1715:   ;
1716:  LBL[26] ;
1717:  R[41]=26    ;
1718:  !RSK gestartet ;
1719:  F[321]=(OFF) ;
1720:  !Sprung zurueck bei Fehler ;
1721:  IF (!F[297] AND !DI[937]),JMP LBL[18] ;
1722:  !STAT EZ2/SP2 FK Fraesen ;
1723:  F[149]=(!F[329]) ;
1724:  DO[116]=(OFF) ;
1725:  DO[162]=(OFF) ;
1726:  R[42]=26    ;
1727:  JMP LBL[1] ;
1728:   ;
1729:   ;
1730:  !************************ ;
1731:  !************************ ;
1732:  !* Fraesen STAT EZ3/SP3 * ;
1733:  !************************ ;
1734:  !************************ ;
1735:   ;
1736:   ;
1737:  !******************************* ;
1738:  !*        Schritt 27           * ;
1739:  !*       STAT EZ3/SP3          * ;
1740:  !* KS3 in Arbeitsst. schwenken * ;
1741:  !******************************* ;
1742:   ;
1743:  LBL[27] ;
1744:  R[41]=27    ;
1745:  !RSK gestartet ;
1746:  F[321]=(OFF) ;
1747:  GO[7]=(31) ;
1748:  GO[9]=(31) ;
1749:  WAIT    .10(sec) ;
1750:  DO[1078]=(F[174]) ;
1751:  DO[1079]=(F[175]) ;
1752:  DO[116]=(ON) ;
1753:  DO[194]=(ON) ;
1754:  DO[1038]=(OFF) ;
1755:  DO[1037]=(!DI[1037]) ;
1756:  DO[18181]=(ON) ;
1757:  WAIT (DI[1037])    ;
1758:  DO[18181]=(OFF) ;
1759:  DO[1037]=(OFF) ;
1760:  !Ueberwachungszeit Grundstellung ;
1761:  TIMER[8]=((-4)) ;
1762:  WAIT ((DI[1162] AND !DI[1163] AND !DI[1164] AND DI[1165]) OR (TIMER[8]>=0))    ;
1763:  F[323]=((TIMER[8]>=0)) ;
1764:  DO[18181]=((TIMER[8]>=0)) ;
1765:  WAIT (DI[1162] AND !DI[1163] AND !DI[1164] AND DI[1165])    ;
1766:  DO[18181]=(OFF) ;
1767:  F[323]=(OFF) ;
1768:  TIMER[8]=((-4)) ;
1769:  DO[1155]=(F[564]) ;
1770:  WAIT ((DI[1155] AND F[564]) OR (!DI[1155] AND !F[564]) OR (TIMER[8]>=0))    ;
1771:  F[323]=((TIMER[8]>=0)) ;
1772:  DO[18181]=((TIMER[8]>=0)) ;
1773:  WAIT ((DI[1155] AND F[564]) OR (!DI[1155] AND !F[564]))    ;
1774:  DO[18181]=(OFF) ;
1775:  F[323]=(OFF) ;
1776:  !Ueberwachungszeit KS3 Schwenken ;
1777:  TIMER[8]=((-4)) ;
1778:  DO[3974]=(ON) ;
1779:  WAIT (DI[1161] OR (TIMER[8]>=0))    ;
1780:  DO[18181]=((TIMER[8]>=0)) ;
1781:  WAIT (DI[1161])    ;
1782:  TIMER[8]=((-6)) ;
1783:  DO[18181]=(OFF) ;
1784:  WAIT ((!DI[1162] AND DI[1163] AND DI[1164] AND !DI[1165]) OR (TIMER[8]>=0))    ;
1785:  F[324]=((TIMER[8]>=0)) ;
1786:  DO[3974]=(OFF) ;
1787:  DO[18181]=((TIMER[8]>=0)) ;
1788:  WAIT ((!DI[1162] AND DI[1163] AND DI[1164] AND !DI[1165]) OR DI[26])    ;
1789:  DO[18181]=(OFF) ;
1790:  F[324]=(OFF) ;
1791:  !Sprung zurueck bei KS3 Fehler ;
1792:  IF (TIMER[8]>=0),JMP LBL[27] ;
1793:  DO[1155]=(OFF) ;
1794:  TIMER[11]=((R[24])) ;
1795:  WAIT ((TIMER[11]>=0) OR !F[564])    ;
1796:  TIMER[11]=STOP ;
1797:  DO[18181]=(ON) ;
1798:  WAIT ((F[184] AND F[174]) OR (F[184] AND F[175]))    ;
1799:  DO[18181]=(OFF) ;
1800:  !Anwahl Startfraesen ;
1801:  IF (!DI[1162] AND DI[1163] AND F[184] AND F[174] AND !F[301]),R[41]=28 ;
1802:  !Anwahl Normalfraesen ;
1803:  IF (!DI[1162] AND DI[1163] AND F[184] AND (F[175] OR F[301])),R[41]=30 ;
1804:  R[42]=27    ;
1805:  JMP LBL[R[41]] ;
1806:   ;
1807:  !************************** ;
1808:  !*       Schritt 28       * ;
1809:  !* STAT EZ3/SP3 SF Teil 1 * ;
1810:  !************************** ;
1811:   ;
1812:  LBL[28] ;
1813:  R[41]=28    ;
1814:  !RSK gestartet ;
1815:  F[321]=(OFF) ;
1816:  F[329]=(OFF) ;
1817:  F[325]=(OFF) ;
1818:  DO[1038]=(OFF) ;
1819:  DO[1037]=(!DI[1037]) ;
1820:  DO[18181]=(ON) ;
1821:  WAIT (DI[1037])    ;
1822:  DO[1037]=(OFF) ;
1823:  DO[18181]=(OFF) ;
1824:  DO[1154]=(ON) ;
1825:  !Warte Fraeser laeuft ;
1826:  TIMER[7]=((-3)) ;
1827:  WAIT (!DI[1154] OR (TIMER[7]>=0))    ;
1828:  WAIT (DI[1154] OR (TIMER[7]>=0))    ;
1829:  F[322]=((TIMER[7]>=0)) ;
1830:  DO[18181]=(ON) ;
1831:  WAIT (!DI[1154])    ;
1832:  WAIT (DI[1154])    ;
1833:  DO[18181]=(OFF) ;
1834:  F[322]=(OFF) ;
1835:  !EZ3/SP3 schliessen ;
1836:  DO[1038]=(ON) ;
1837:  !Fraeser ausblasen AUS/EIN ;
1838:  DO[1167]=(F[330]) ;
1839:  TIMER[9]=((-4)) ;
1840:  !EZ3/SP3 Kraft erreicht ;
1841:  WAIT ((DI[1038] AND !DI[1092] AND !DI[1100] AND !DI[1094] AND !DI[1095]) OR (TIMER[9]>=0))    ;
1842:  F[325]=((TIMER[9]>=0)) ;
1843:  DO[18181]=(ON) ;
1844:  DO[1038]=((TIMER[9]<0)) ;
1845:  DO[1154]=((TIMER[9]<0)) ;
1846:  WAIT ((DI[1038] AND !DI[1092] AND !DI[1100] AND !DI[1094] AND !DI[1095]) OR DI[26] OR DI[27])    ;
1847:  DO[18181]=(OFF) ;
1848:  !EZ3/SP3 Fehler Kraftaufbau ;
1849:  IF (F[325]),JMP LBL[2801] ;
1850:  TIMER[9]=((-5)) ;
1851:  LBL[2800] ;
1852:  WAIT (!DI[1154] OR F[325] OR (TIMER[9]>=0))    ;
1853:  WAIT (DI[1154] OR F[325] OR (TIMER[9]>=0))    ;
1854:  R[1]=(R[1]+1) ;
1855:  F[329]=((TIMER[9]>=0)) ;
1856:  !Fraeszeit ueberschritten ;
1857:  IF (F[329]),JMP LBL[2801] ;
1858:  !Umdrehungen Vergleichen ;
1859:  IF (R[1]<R[17]),JMP LBL[2800] ;
1860:  F[186]=(ON) ;
1861:  LBL[2801] ;
1862:  DO[1154]=((TIMER[9]<0)) ;
1863:  !Fraeser ausblasen EIN ;
1864:  DO[1167]=(F[330] OR (TIMER[9]<0)) ;
1865:  DO[1038]=(OFF) ;
1866:  !EZ3/SP3 oeffnen ;
1867:  DO[1037]=(!DI[1037]) ;
1868:  DO[18181]=(F[329]) ;
1869:  WAIT (!F[329] OR DI[26] OR DI[27])    ;
1870:  DO[18181]=(OFF) ;
1871:  DO[18181]=(ON) ;
1872:  WAIT (DI[1037])    ;
1873:  DO[18181]=(OFF) ;
1874:  DO[1037]=(OFF) ;
1875:  !Umdrehungen ruecksetzen ;
1876:  R[1]=0    ;
1877:  R[42]=28    ;
1878:  IF (F[329] OR F[325]),JMP LBL[28] ;
1879:  JMP LBL[29] ;
1880:   ;
1881:  !************************** ;
1882:  !*      Schritt 29        * ;
1883:  !* STAT EZ3/SP3 SF Teil 2 * ;
1884:  !************************** ;
1885:   ;
1886:  LBL[29] ;
1887:  R[41]=29    ;
1888:  !RSK gestartet ;
1889:  F[321]=(OFF) ;
1890:  F[329]=(OFF) ;
1891:  F[325]=(OFF) ;
1892:  DO[1038]=(OFF) ;
1893:  DO[1037]=(!DI[1037]) ;
1894:  DO[18181]=(ON) ;
1895:  WAIT (DI[1037])    ;
1896:  DO[18181]=(OFF) ;
1897:  DO[1154]=(ON) ;
1898:  DO[1037]=(OFF) ;
1899:  !EZ3/SP3 schliessen ;
1900:  DO[1038]=(ON) ;
1901:  !Fraeser ausblasen AUS/EIN ;
1902:  DO[1167]=(F[330]) ;
1903:  TIMER[9]=((-4)) ;
1904:  !EZ3/SP3 Kraft erreicht ;
1905:  WAIT ((DI[1038] AND !DI[1092] AND !DI[1100] AND !DI[1094] AND !DI[1095]) OR (TIMER[9]>=0))    ;
1906:  F[325]=((TIMER[9]>=0)) ;
1907:  DO[18181]=(ON) ;
1908:  DO[1038]=((TIMER[9]<0)) ;
1909:  DO[1154]=((TIMER[9]<0)) ;
1910:  WAIT ((DI[1038] AND !DI[1092] AND !DI[1100] AND !DI[1094] AND !DI[1095]) OR DI[26] OR DI[27])    ;
1911:  DO[18181]=(OFF) ;
1912:  !EZ3/SP3 Fehler Kraftaufbau ;
1913:  IF (F[325]),JMP LBL[2901] ;
1914:  TIMER[9]=((-5)) ;
1915:  LBL[2900] ;
1916:  WAIT (!DI[1154] OR F[325] OR (TIMER[9]>=0))    ;
1917:  WAIT (DI[1154] OR F[325] OR (TIMER[9]>=0))    ;
1918:  R[1]=(R[1]+1) ;
1919:  F[329]=((TIMER[9]>=0)) ;
1920:  !Fraeszeit ueberschritten ;
1921:  IF (F[329]),JMP LBL[2901] ;
1922:  !Umdrehungen Vergleichen ;
1923:  IF (R[1]<R[18]),JMP LBL[2900] ;
1924:  F[188]=(ON) ;
1925:  LBL[2901] ;
1926:  DO[1154]=((TIMER[9]<0)) ;
1927:  !Fraeser ausblasen EIN ;
1928:  DO[1167]=PULSE,4.0sec ;
1929:  DO[1038]=(OFF) ;
1930:  !EZ3/SP3 oeffnen ;
1931:  DO[1037]=(!DI[1037]) ;
1932:  DO[18181]=(F[329]) ;
1933:  WAIT (!F[329] OR DI[26] OR DI[27])    ;
1934:  DO[18181]=(OFF) ;
1935:  DO[18181]=(ON) ;
1936:  WAIT (DI[1037])    ;
1937:  DO[18181]=(OFF) ;
1938:  DO[1037]=(OFF) ;
1939:  !Umdrehungen ruecksetzen ;
1940:  R[1]=0    ;
1941:  R[42]=29    ;
1942:  IF (F[329] OR F[325]),JMP LBL[29] ;
1943:  JMP LBL[31] ;
1944:   ;
1945:  !******************* ;
1946:  !*   Schritt 30    * ;
1947:  !* STAT EZ3/SP3 NF * ;
1948:  !******************* ;
1949:   ;
1950:  LBL[30] ;
1951:  R[41]=30    ;
1952:  !RSK gestartet ;
1953:  F[321]=(OFF) ;
1954:  F[329]=(OFF) ;
1955:  F[325]=(OFF) ;
1956:  !Zähler wegspeichern für 2ten Hub ;
1957:  R[45]=(R[19]) ;
1958:  IF (F[190] AND F[732]),R[19]=(R[38]) ;
1959:  DO[1038]=(OFF) ;
1960:  DO[1037]=(!DI[1037]) ;
1961:  DO[18181]=(ON) ;
1962:  WAIT (DI[1037])    ;
1963:  DO[18181]=(OFF) ;
1964:  DO[1154]=(ON) ;
1965:  DO[1037]=(OFF) ;
1966:  !EZ3/SP3 schliessen ;
1967:  DO[1038]=(ON) ;
1968:  !Fraeser ausblasen AUS ;
1969:  DO[1167]=(F[330]) ;
1970:  TIMER[9]=((-4)) ;
1971:  !EZ3/SP3 Kraft erreicht ;
1972:  WAIT ((DI[1038] AND !DI[1092] AND !DI[1100] AND !DI[1094] AND !DI[1095]) OR (TIMER[9]>=0))    ;
1973:  F[325]=((TIMER[9]>=0)) ;
1974:  DO[18181]=(ON) ;
1975:  DO[1038]=((TIMER[9]<0)) ;
1976:  DO[1154]=((TIMER[9]<0)) ;
1977:  WAIT ((DI[1038] AND !DI[1092] AND !DI[1100] AND !DI[1094] AND !DI[1095]) OR DI[26] OR DI[27])    ;
1978:  DO[18181]=(OFF) ;
1979:  !EZ3/SP3 Fehler Kraftaufbau ;
1980:  IF (F[325]),JMP LBL[3001] ;
1981:  TIMER[9]=((-5)) ;
1982:  LBL[3000] ;
1983:  WAIT (!DI[1154] OR F[325] OR (TIMER[9]>=0))    ;
1984:  WAIT (DI[1154] OR F[325] OR (TIMER[9]>=0))    ;
1985:  R[1]=(R[1]+1) ;
1986:  F[329]=((TIMER[9]>=0)) ;
1987:  !Fraeszeit ueberschritten ;
1988:  IF (F[329]),JMP LBL[3001] ;
1989:  !Umdrehungen Vergleichen ;
1990:  IF (R[1]<R[19]),JMP LBL[3000] ;
1991:  !EZ3/SP3 2 Huebe bei NF ;
1992:  IF (!F[200]),JMP LBL[3001] ;
1993:  IF (F[190]),F[188]=(ON) ;
1994:  F[190]=(ON) ;
1995:  LBL[3001] ;
1996:  DO[1154]=((TIMER[9]<0)) ;
1997:  !Fraeser ausblasen EIN ;
1998:  DO[1167]=PULSE,4.0sec ;
1999:  !EZ3/SP3 oeffnen ;
2000:  DO[1038]=(OFF) ;
2001:  DO[1037]=(!DI[1037]) ;
2002:  DO[18181]=(F[329]) ;
2003:  WAIT (!F[329] OR DI[26] OR DI[27])    ;
2004:  DO[18181]=(OFF) ;
2005:  DO[18181]=(ON) ;
2006:  WAIT (DI[1037])    ;
2007:  DO[18181]=(OFF) ;
2008:  DO[1037]=(OFF) ;
2009:  !Umdrehungen ruecksetzen ;
2010:  R[1]=0    ;
2011:  R[42]=30    ;
2012:  IF (F[190] AND F[732]),GO[3]=36 ;
2013:  IF (F[188] AND F[732]),R[19]=(R[45]) ;
2014:  IF (F[329] OR F[325] OR (!F[188] AND F[200])),JMP LBL[30] ;
2015:  F[190]=(ON) ;
2016:  JMP LBL[31] ;
2017:   ;
2018:  !**************************** ;
2019:  !*        Schritt 31        * ;
2020:  !* STAT EZ3/SP3 i.O./n.i.O. * ;
2021:  !**************************** ;
2022:   ;
2023:  LBL[31] ;
2024:  R[41]=31    ;
2025:  !Fraesueberwachung starten ;
2026:  TIMER[7]=((-5)) ;
2027:  WAIT ((F[174] OR F[175]) AND (F[190] OR (F[186] AND F[188])) OR (TIMER[7]>=0))    ;
2028:  F[329]=((TIMER[7]>=0)) ;
2029:  IF (!F[329]),R[41]=32 ;
2030:  IF (F[329]),R[41]=30 ;
2031:  !KF1 U-Merker ruecksetzen ;
2032:  F[186]=(OFF) ;
2033:  F[188]=(OFF) ;
2034:  F[190]=(OFF) ;
2035:  R[42]=31    ;
2036:  JMP LBL[R[41]] ;
2037:   ;
2038:  !**************************** ;
2039:  !*       Schritt 32         * ;
2040:  !*      STAT EZ3/SP3        * ;
2041:  !* KS3 in Ruhest. schwenken * ;
2042:  !**************************** ;
2043:   ;
2044:  LBL[32] ;
2045:  R[41]=32    ;
2046:  !RSK gestartet ;
2047:  F[321]=(OFF) ;
2048:  DO[1038]=(OFF) ;
2049:  DO[1037]=(!DI[1037]) ;
2050:  DO[18181]=(ON) ;
2051:  WAIT (DI[1037])    ;
2052:  DO[18181]=(OFF) ;
2053:  DO[1037]=(OFF) ;
2054:  TIMER[8]=((-4)) ;
2055:  WAIT ((DI[1164] AND !DI[1162] AND !DI[1165] AND DI[1163]) OR (TIMER[8]>=0))    ;
2056:  F[324]=((TIMER[8]>=0)) ;
2057:  DO[18181]=((TIMER[8]>=0)) ;
2058:  WAIT (DI[1164] AND !DI[1162] AND !DI[1165] AND DI[1163])    ;
2059:  DO[18181]=(OFF) ;
2060:  F[324]=(OFF) ;
2061:  TIMER[8]=((-4)) ;
2062:  DO[1155]=(F[564]) ;
2063:  WAIT ((DI[1155] AND F[564]) OR (!DI[1155] AND !F[564]) OR (TIMER[8]>=0))    ;
2064:  F[323]=((TIMER[8]>=0)) ;
2065:  DO[18181]=((TIMER[8]>=0)) ;
2066:  WAIT ((DI[1155] AND F[564]) OR (!DI[1155] AND !F[564]))    ;
2067:  DO[18181]=(OFF) ;
2068:  F[323]=(OFF) ;
2069:  !Ueberwachungszeit KS3 Schwenken ;
2070:  TIMER[8]=((-4)) ;
2071:  DO[3971]=(ON) ;
2072:  WAIT (DI[1161] OR (TIMER[8]>=0))    ;
2073:  DO[18181]=((TIMER[8]>=0)) ;
2074:  WAIT (DI[1161])    ;
2075:  TIMER[8]=((-6)) ;
2076:  DO[18181]=(OFF) ;
2077:  WAIT ((!DI[1164] AND DI[1162] AND DI[1165] AND !DI[1163]) OR (TIMER[8]>=0))    ;
2078:  F[323]=((TIMER[8]>=0)) ;
2079:  DO[3971]=(OFF) ;
2080:  DO[18181]=((TIMER[8]>=0)) ;
2081:  WAIT ((!DI[1164] AND DI[1162] AND DI[1165] AND !DI[1163]) OR DI[26])    ;
2082:  DO[18181]=(OFF) ;
2083:  F[323]=(OFF) ;
2084:  DO[1154]=(OFF) ;
2085:  DO[1155]=(OFF) ;
2086:  !Sprung zurueck bei KS3 Fehler ;
2087:  IF (TIMER[8]>=0),JMP LBL[32] ;
2088:  R[42]=32    ;
2089:  JMP LBL[33] ;
2090:   ;
2091:  !*********************** ;
2092:  !*     Schritt 33      * ;
2093:  !*    STAT EZ3/SP3     * ;
2094:  !* Messen nach Fraesen * ;
2095:  !*********************** ;
2096:   ;
2097:  LBL[33] ;
2098:  R[41]=33    ;
2099:  !RSK gestartet ;
2100:  F[321]=(OFF) ;
2101:  GO[9]=1 ;
2102:  WAIT    .10(sec) ;
2103:  DO[1106]=(ON) ;
2104:  !STAT EZ3/SP3 FK Fraesen ;
2105:  DO[18181]=(ON) ;
2106:  WAIT (!DI[1106] AND DI[1107] AND !DI[1108])    ;
2107:  DO[18181]=(OFF) ;
2108:  DO[1106]=(OFF) ;
2109:  GO[7]=(31) ;
2110:  GO[9]=(31) ;
2111:  WAIT    .10(sec) ;
2112:  DO[1077]=(ON) ;
2113:  TIMER[9]=((-8)) ;
2114:  WAIT (DI[1077] OR (TIMER[9]>=0))    ;
2115:  DO[326]=((TIMER[9]>=0)) ;
2116:  DO[18181]=(ON) ;
2117:  WAIT (DI[1077] OR DI[26] OR DI[27])    ;
2118:  DO[18181]=(OFF) ;
2119:  DO[326]=(OFF) ;
2120:  F[179]=(DI[1096] OR DI[1097]) ;
2121:  DO[1077]=(OFF) ;
2122:  F[180]=(DI[1056] OR (DI[1055] AND DI[1054] AND DI[1053])) ;
2123:  TIMER[7]=((-2)) ;
2124:  WAIT ((!F[180] AND !F[179]) OR (TIMER[7]>=0))    ;
2125:  F[329]=((TIMER[7]>=0)) ;
2126:  DO[18181]=(F[329]) ;
2127:  WAIT ((!F[180] AND !F[179]) OR DI[26] OR DI[27])    ;
2128:  DO[18181]=(OFF) ;
2129:  F[329]=(OFF) ;
2130:  F[298]=(F[180] OR F[179]) ;
2131:  DO[1037]=(!DI[1037]) ;
2132:  DO[18181]=(ON) ;
2133:  WAIT ((DI[1037] AND !DI[1104]) OR (DI[1037] AND F[298]))    ;
2134:  DO[18181]=(OFF) ;
2135:  DO[1037]=(OFF) ;
2136:  R[42]=33    ;
2137:  !EZ3/SP3 wiederh. bei Messfehler ;
2138:  IF (F[298]),JMP LBL[27] ;
2139:  DO[1078]=(OFF) ;
2140:  DO[1079]=(OFF) ;
2141:  !KS nicht bei K-Verschleiss ;
2142:  IF (DI[1097]),JMP LBL[35] ;
2143:  !EZ3/SP3 2.Setzhub nach Fraesen ;
2144:  IF (F[335] AND F[174]),JMP LBL[57] ;
2145:  !EZ3/SP3 Kurzschluss schweissen ;
2146:  IF (F[335] AND !F[174]),JMP LBL[34] ;
2147:  !EZ3/SP3 Kurzschluss schweissen ;
2148:  IF (!F[335]),JMP LBL[34] ;
2149:   ;
2150:  !************************** ;
2151:  !*      Schritt 34        * ;
2152:  !*     STAT EZ3/SP3       * ;
2153:  !* Kurzschlussschweissung * ;
2154:  !************************** ;
2155:   ;
2156:  LBL[34] ;
2157:  R[41]=34    ;
2158:  !RSK gestartet ;
2159:  F[321]=(OFF) ;
2160:  DO[209]=(ON) ;
2161:  !EZ3/SP3/SK3 Prog. ;
2162:  IF (F[174] AND !F[301]),GO[7]=(41) ;
2163:  IF (F[174] AND !F[301]),GO[9]=(41) ;
2164:  IF (F[175] OR F[301]),GO[7]=(51) ;
2165:  IF (F[175] OR F[301]),GO[9]=(51) ;
2166:  WAIT    .10(sec) ;
2167:  DO[1037]=(OFF) ;
2168:  DO[1038]=(OFF) ;
2169:  DO[1105]=(OFF) ;
2170:  DO[514]=(OFF) ;
2171:  F[176]=(OFF) ;
2172:  F[306]=(OFF) ;
2173:  F[303]=(!DI[1089] AND DI[1104]) ;
2174:  DO[18181]=(ON) ;
2175:  WAIT (DI[1025] AND DI[1033] AND DI[1034] AND (!DI[1104] OR (DI[1089] AND DI[1104])))    ;
2176:  DO[18181]=(OFF) ;
2177:  F[303]=(OFF) ;
2178:  DO[18181]=(ON) ;
2179:  WAIT ((!DI[1105] AND DI[1112] AND DI[1122] AND !F[176]) OR (!DI[1112] AND DI[1122] AND DI[209]))    ;
2180:  DO[18181]=(OFF) ;
2181:  !EZ3/SP3 schliessen ;
2182:  DO[1038]=(ON) ;
2183:  TIMER[9]=((-4)) ;
2184:  !EZ3/SP3 Kraft erreicht ;
2185:  WAIT ((DI[1038] AND !DI[1092] AND !DI[1100]) OR DI[1094] OR DI[1095] OR (TIMER[9]>=0))    ;
2186:  DO[1038]=(DI[1038] AND !DI[1094] AND !DI[1095]) ;
2187:  DO[1037]=(!DO[1038]) ;
2188:  !Schweissen START ;
2189:  DO[1105]=(DI[1038] AND !DI[1094] AND !DI[1095]) ;
2190:  !EZ3/SP3 Fehler Ausgleich ;
2191:  F[302]=(DI[1038] AND DI[1039]) ;
2192:  !EZ3/SP3 Fehler SZ ;
2193:  F[300]=(DI[1094] OR DI[1095]) ;
2194:  !SK3 FK ;
2195:  TIMER[9]=((-10)) ;
2196:  WAIT ((F[176] AND DO[1105]) OR ((DI[1124] OR DI[1125]) AND (DI[1105] AND DO[1105])) OR (DI[1091] AND DI[1104]) OR !DO[1105] OR (TIMER[9]>=0))    ;
2197:  F[297]=(F[176] OR (DI[1124] AND !DI[1126] AND !DI[1095] AND DI[1105])) ;
2198:  !SK3 Fehler ;
2199:  F[301]=(!F[297] AND !F[298] AND DO[1105]) ;
2200:  DO[1105]=(OFF) ;
2201:  DO[1038]=(OFF) ;
2202:  DO[18181]=(ON) ;
2203:  F[749]=(!F[297] AND !F[748]) ;
2204:  F[748]=(!F[297]) ;
2205:  WAIT (F[297] OR DI[26] OR DI[27] OR (F[749] AND F[731]))    ;
2206:  WAIT (!DI[26] AND !DI[27])    ;
2207:  DO[18181]=(OFF) ;
2208:  !EZ3/SP3 oeffnen ;
2209:  DO[1037]=(!DI[1037]) ;
2210:  DO[18181]=(ON) ;
2211:  WAIT (DI[1037])    ;
2212:  DO[18181]=(OFF) ;
2213:  DO[1037]=(OFF) ;
2214:  F[303]=(OFF) ;
2215:  DO[209]=(OFF) ;
2216:  R[42]=34    ;
2217:  JMP LBL[35] ;
2218:   ;
2219:  !************************** ;
2220:  !*       Schritt 35       * ;
2221:  !*      STAT EZ3/SP3      * ;
2222:  !************************** ;
2223:   ;
2224:  LBL[35] ;
2225:  R[41]=35    ;
2226:  !RSK gestartet ;
2227:  F[321]=(OFF) ;
2228:  !Sprung zurueck bei Fehler ;
2229:  IF (!F[297] AND !DI[1097]),JMP LBL[27] ;
2230:  !STAT EZ3/SP3 FK Fraesen ;
2231:  F[185]=(!F[329]) ;
2232:  DO[116]=(OFF) ;
2233:  DO[194]=(OFF) ;
2234:  R[42]=35    ;
2235:  JMP LBL[1] ;
2236:   ;
2237:   ;
2238:  !***************** ;
2239:  !***************** ;
2240:  !* MS1 Reinigung * ;
2241:  !***************** ;
2242:  !***************** ;
2243:   ;
2244:   ;
2245:  !******************************* ;
2246:  !*         Schritt 36          * ;
2247:  !*       MS1 Reinigung         * ;
2248:  !* KS3 in Arbeitsst. schwenken * ;
2249:  !******************************* ;
2250:   ;
2251:  LBL[36] ;
2252:  R[41]=36    ;
2253:  !RSK gestartet ;
2254:  F[321]=(OFF) ;
2255:  !MS bei Reinigung ;
2256:  DO[116]=(ON) ;
2257:  !Reinigung MS1 gestartet ;
2258:  F[604]=(ON) ;
2259:  !Ueberwachungszeit KS3 ;
2260:  TIMER[8]=((-4)) ;
2261:  WAIT ((!DI[1164] AND DI[1162] AND DI[1165] AND !DI[1163]) OR (TIMER[8]>=0))    ;
2262:  F[323]=((TIMER[8]>=0)) ;
2263:  DO[18181]=((TIMER[8]>=0)) ;
2264:  WAIT (!DI[1164] AND DI[1162] AND DI[1165] AND !DI[1163])    ;
2265:  DO[18181]=(OFF) ;
2266:  F[323]=(OFF) ;
2267:  !KS3 in Arbeitsst. schwenken ;
2268:  TIMER[8]=((-4)) ;
2269:  DO[3974]=(ON) ;
2270:  WAIT (DI[1161] OR (TIMER[8]>=0))    ;
2271:  DO[18181]=((TIMER[8]>=0)) ;
2272:  WAIT (DI[1161])    ;
2273:  DO[18181]=(OFF) ;
2274:  TIMER[8]=((-6)) ;
2275:  WAIT ((DI[1164] AND !DI[1162] AND !DI[1165] AND DI[1163]) OR (TIMER[8]>=0))    ;
2276:  F[324]=((TIMER[8]>=0)) ;
2277:  DO[3974]=(OFF) ;
2278:  DO[18181]=((TIMER[8]>=0)) ;
2279:  WAIT ((DI[1164] AND !DI[1162] AND !DI[1165] AND DI[1163]) OR DI[26])    ;
2280:  DO[18181]=(OFF) ;
2281:  F[324]=(OFF) ;
2282:  !Sprung bei Fehler KS3 schwenken ;
2283:  IF (TIMER[8]>=0),JMP LBL[36] ;
2284:  R[42]=36    ;
2285:  JMP LBL[37] ;
2286:   ;
2287:  !*************************** ;
2288:  !*      Schritt 37         * ;
2289:  !* MS1 Reinigung starten   * ;
2290:  !*************************** ;
2291:   ;
2292:  LBL[37] ;
2293:  R[41]=37    ;
2294:  TIMER[9]=((-2)) ;
2295:  WAIT ((DI[10] AND DI[13] AND DI[23]) OR (TIMER[9]>=0))    ;
2296:  F[329]=((TIMER[9]>=0)) ;
2297:  DO[18181]=((TIMER[9]>=0)) ;
2298:  WAIT (DI[10] AND DI[13] AND DI[23])    ;
2299:  F[329]=(OFF) ;
2300:  DO[18181]=(OFF) ;
2301:  !MS1 Reinigung i.O. ;
2302:  DO[18181]=(ON) ;
2303:  WAIT (DI[1864])    ;
2304:  DO[18181]=(OFF) ;
2305:  !MS1 Ausblasen EIN ;
2306:  DO[1870]=(ON) ;
2307:  !MS1 Reinigung EIN ;
2308:  TIMER[9]=((-1)) ;
2309:  DO[1864]=(ON) ;
2310:  !Einschaltdauer Reingung ;
2311:  TIMER[7]=((R[26])) ;
2312:  WAIT (!DI[1864] OR (TIMER[9]>=0))    ;
2313:  F[329]=((TIMER[9]>=0)) ;
2314:  DO[18181]=((TIMER[9]>=0)) ;
2315:  WAIT (!DI[1864] OR DI[26])    ;
2316:  WAIT ((TIMER[7]>=0))    ;
2317:  F[329]=(OFF) ;
2318:  DO[18181]=(OFF) ;
2319:  !MS1 Reinigung AUS ;
2320:  DO[1864]=(OFF) ;
2321:  TIMER[9]=((-6)) ;
2322:  WAIT (DI[1864] OR (TIMER[9]>=0))    ;
2323:  F[329]=((TIMER[9]>=0)) ;
2324:  DO[18181]=((TIMER[9]>=0)) ;
2325:  WAIT (DI[1864] OR DI[26] OR !DI[13] OR !DI[23])    ;
2326:  IF (DI[26] OR !DI[13] OR !DI[23]),JMP LBL[37] ;
2327:  F[329]=(OFF) ;
2328:  DO[18181]=(OFF) ;
2329:  !MS1 Ausblasen AUS ;
2330:  DO[1870]=(OFF) ;
2331:  !MS1 Einspruehen ;
2332:  TIMER[9]=((R[23])) ;
2333:  DO[520]=(!F[574] AND F[575]) ;
2334:  DO[1871]=(F[574] AND F[575]) ;
2335:  WAIT (!F[575] OR (TIMER[9]>=0))    ;
2336:  DO[520]=(OFF) ;
2337:  DO[1871]=(OFF) ;
2338:  R[42]=37    ;
2339:  JMP LBL[38] ;
2340:   ;
2341:  !**************************** ;
2342:  !*          Schritt 38      * ;
2343:  !*       MS1 Reinigung      * ;
2344:  !* KS3 in Ruhest. schwenken * ;
2345:  !**************************** ;
2346:   ;
2347:  LBL[38] ;
2348:  R[41]=38    ;
2349:  !Ueberwachungszeit KS3 ;
2350:  TIMER[8]=((-4)) ;
2351:  WAIT ((DI[1164] AND !DI[1162] AND !DI[1165] AND DI[1163]) OR (TIMER[8]>=0))    ;
2352:  F[324]=((TIMER[8]>=0)) ;
2353:  DO[18181]=((TIMER[8]>=0)) ;
2354:  WAIT (DI[1164] AND !DI[1162] AND !DI[1165] AND DI[1163])    ;
2355:  DO[18181]=(OFF) ;
2356:  F[324]=(OFF) ;
2357:  !KS3 in Ruhestest. schwenken ;
2358:  TIMER[8]=((-4)) ;
2359:  DO[3971]=(ON) ;
2360:  WAIT (DI[1161] OR (TIMER[8]>=0))    ;
2361:  DO[18181]=((TIMER[8]>=0)) ;
2362:  WAIT (DI[1161])    ;
2363:  DO[18181]=(OFF) ;
2364:  TIMER[8]=((-6)) ;
2365:  WAIT ((!DI[1164] AND DI[1162] AND DI[1165] AND !DI[1163]) OR (TIMER[8]>=0))    ;
2366:  F[323]=((TIMER[8]>=0)) ;
2367:  DO[3971]=(OFF) ;
2368:  DO[18181]=((TIMER[8]>=0)) ;
2369:  WAIT ((!DI[1164] AND DI[1162] AND DI[1165] AND !DI[1163]) OR DI[26])    ;
2370:  DO[18181]=(OFF) ;
2371:  F[323]=(OFF) ;
2372:  !Sprung bei Fehler KS3 schwenken ;
2373:  IF (TIMER[8]>=0),JMP LBL[38] ;
2374:  R[42]=38    ;
2375:  JMP LBL[39] ;
2376:   ;
2377:  !***************************** ;
2378:  !*         Schritt 39        * ;
2379:  !* MS1 Reinigung ruecksetzen * ;
2380:  !***************************** ;
2381:   ;
2382:  LBL[39] ;
2383:  R[41]=39    ;
2384:  !MS1 Zaehler ruecksetzen ;
2385:  R[21]=0    ;
2386:  !MS FRG Reinigung ;
2387:  F[603]=(OFF) ;
2388:  !MS1 Reinigung FK ;
2389:  F[605]=(ON) ;
2390:  R[42]=39    ;
2391:  JMP LBL[1] ;
2392:   ;
2393:   ;
2394:  !***************** ;
2395:  !***************** ;
2396:  !* MS2 Reinigung * ;
2397:  !***************** ;
2398:  !***************** ;
2399:   ;
2400:   ;
2401:  !******************************* ;
2402:  !*         Schritt 40          * ;
2403:  !*       MS2 Reinigung         * ;
2404:  !* KS2 in Arbeitsst. schwenken * ;
2405:  !******************************* ;
2406:   ;
2407:  LBL[40] ;
2408:  R[41]=40    ;
2409:  !RSK gestartet ;
2410:  F[321]=(OFF) ;
2411:  !Reinigung MS2 gestartet ;
2412:  F[608]=(ON) ;
2413:  !MS bei Reinigung ;
2414:  DO[116]=(ON) ;
2415:  !Ueberwachungszeit KS2 ;
2416:  TIMER[8]=((-4)) ;
2417:  WAIT ((!DI[1004] AND DI[1002] AND DI[1005] AND !DI[1003]) OR (TIMER[8]>=0))    ;
2418:  F[323]=((TIMER[8]>=0)) ;
2419:  DO[18181]=((TIMER[8]>=0)) ;
2420:  WAIT (!DI[1004] AND DI[1002] AND DI[1005] AND !DI[1003])    ;
2421:  DO[18181]=(OFF) ;
2422:  F[323]=(OFF) ;
2423:  !KS2 in Arbeitsst. schwenken ;
2424:  TIMER[8]=((-4)) ;
2425:  DO[3973]=(ON) ;
2426:  WAIT (DI[1001] OR (TIMER[8]>=0))    ;
2427:  DO[18181]=((TIMER[8]>=0)) ;
2428:  WAIT (DI[1001])    ;
2429:  DO[18181]=(OFF) ;
2430:  TIMER[8]=((-4)) ;
2431:  WAIT ((DI[1004] AND !DI[1002] AND !DI[1005] AND DI[1003]) OR (TIMER[8]>=0))    ;
2432:  F[324]=((TIMER[8]>=0)) ;
2433:  DO[3973]=(OFF) ;
2434:  DO[18181]=((TIMER[8]>=0)) ;
2435:  WAIT ((DI[1004] AND !DI[1002] AND !DI[1005] AND DI[1003]) OR DI[26])    ;
2436:  DO[18181]=(OFF) ;
2437:  F[324]=(OFF) ;
2438:  !Sprung bei Fehler KS2 schwenken ;
2439:  IF (TIMER[8]>=0),JMP LBL[40] ;
2440:  R[42]=40    ;
2441:  JMP LBL[41] ;
2442:   ;
2443:  !*************************** ;
2444:  !*      Schritt 41         * ;
2445:  !* MS2 Reinigung starten   * ;
2446:  !*************************** ;
2447:   ;
2448:  LBL[41] ;
2449:  R[41]=41    ;
2450:  TIMER[9]=((-2)) ;
2451:  WAIT ((DI[10] AND DI[13] AND DI[23]) OR (TIMER[9]>=0))    ;
2452:  F[329]=((TIMER[9]>=0)) ;
2453:  DO[18181]=((TIMER[9]>=0)) ;
2454:  WAIT (DI[10] AND DI[13] AND DI[23])    ;
2455:  F[329]=(OFF) ;
2456:  DO[18181]=(OFF) ;
2457:  !MS2 Ausblasen EIN ;
2458:  DO[1902]=(ON) ;
2459:  !MS2 Reinigung EIN ;
2460:  TIMER[9]=((-1)) ;
2461:  DO[1896]=(ON) ;
2462:  WAIT (!DI[1896] OR (TIMER[9]>=0))    ;
2463:  F[329]=((TIMER[9]>=0)) ;
2464:  DO[18181]=((TIMER[9]>=0)) ;
2465:  WAIT (!DI[1896] OR DI[26])    ;
2466:  F[329]=(OFF) ;
2467:  DO[18181]=(OFF) ;
2468:  !MS2 Reinigung AUS ;
2469:  DO[1896]=(OFF) ;
2470:  TIMER[9]=((-6)) ;
2471:  WAIT (DI[1896] OR (TIMER[9]>=0))    ;
2472:  F[329]=((TIMER[9]>=0)) ;
2473:  DO[18181]=((TIMER[9]>=0)) ;
2474:  WAIT (DI[1896] OR DI[26] OR !DI[13] OR !DI[23])    ;
2475:  IF (DI[26] OR !DI[13] OR !DI[23]),JMP LBL[41] ;
2476:  F[329]=(OFF) ;
2477:  DO[18181]=(OFF) ;
2478:  !MS2 Ausblasen AUS ;
2479:  DO[1902]=(OFF) ;
2480:  !MS2 Einspruehen ;
2481:  TIMER[9]=((R[23])) ;
2482:  DO[528]=(!F[583] AND F[584]) ;
2483:  DO[1903]=(F[583] AND F[585]) ;
2484:  WAIT (!F[584] OR (TIMER[9]>=0))    ;
2485:  DO[528]=(OFF) ;
2486:  DO[1903]=(OFF) ;
2487:  R[42]=41    ;
2488:  JMP LBL[42] ;
2489:   ;
2490:  !**************************** ;
2491:  !*          Schritt 42      * ;
2492:  !*       MS2 Reinigung      * ;
2493:  !* KS2 in Ruhest. schwenken * ;
2494:  !**************************** ;
2495:   ;
2496:  LBL[42] ;
2497:  R[41]=42    ;
2498:  !Ueberwachungszeit KS2 ;
2499:  TIMER[8]=((-4)) ;
2500:  WAIT ((DI[1004] AND !DI[1002] AND !DI[1005] AND DI[1003]) OR (TIMER[8]>=0))    ;
2501:  F[324]=((TIMER[8]>=0)) ;
2502:  DO[18181]=((TIMER[8]>=0)) ;
2503:  WAIT (DI[1004] AND !DI[1002] AND !DI[1005] AND DI[1003])    ;
2504:  DO[18181]=(OFF) ;
2505:  F[324]=(OFF) ;
2506:  !KS2 in Ruhestest. schwenken ;
2507:  TIMER[8]=((-4)) ;
2508:  DO[3970]=(ON) ;
2509:  WAIT (DI[1001] OR (TIMER[8]>=0))    ;
2510:  DO[18181]=((TIMER[8]>=0)) ;
2511:  WAIT (DI[1001])    ;
2512:  DO[18181]=(OFF) ;
2513:  TIMER[8]=((-6)) ;
2514:  WAIT ((!DI[1004] AND DI[1002] AND DI[1005] AND !DI[1003]) OR (TIMER[8]>=0))    ;
2515:  F[323]=((TIMER[8]>=0)) ;
2516:  DO[3970]=(OFF) ;
2517:  DO[18181]=((TIMER[8]>=0)) ;
2518:  WAIT ((!DI[1004] AND DI[1002] AND DI[1005] AND !DI[1003]) OR DI[26])    ;
2519:  DO[18181]=(OFF) ;
2520:  F[323]=(OFF) ;
2521:  !Sprung bei Fehler KS2 schwenken ;
2522:  IF (TIMER[8]>=0),JMP LBL[42] ;
2523:  R[42]=42    ;
2524:  JMP LBL[43] ;
2525:   ;
2526:  !***************************** ;
2527:  !*         Schritt 43        * ;
2528:  !* MS2 Reinigung ruecksetzen * ;
2529:  !***************************** ;
2530:   ;
2531:  LBL[43] ;
2532:  R[41]=43    ;
2533:  !MS2 Zaehler ruecksetzen ;
2534:  R[22]=0    ;
2535:  !MS2 FRG Reinigung ;
2536:  F[607]=(OFF) ;
2537:  !MS2 Reinigung FK ;
2538:  F[609]=(ON) ;
2539:  R[42]=43    ;
2540:  JMP LBL[1] ;
2541:   ;
2542:  !******************************** ;
2543:  !*            Schritt 44 ;
2544:  !*          KL1 Spueleimer ;
2545:  !*  (an Pneum. Schwenkeinheit KL1 ;
2546:  !*     KL1 in Arbeitsst. schwenke ;
2547:  !******************************** ;
2548:   ;
2549:  LBL[44] ;
2550:  R[41]=44    ;
2551:  !RSK gestartet ;
2552:  F[321]=(OFF) ;
2553:  DO[161]=(ON) ;
2554:  !Steuerluft EIN ;
2555:  DO[2113]=(ON) ;
2556:  TIMER[9]=((-2)) ;
2557:  !Warte auf Vorwahl Ventilinsel ;
2558:  WAIT ((F[523] AND !F[524]) OR (!F[523] AND F[524]) OR (TIMER[9]>=0))    ;
2559:  DO[120]=(TIMER[9]>=0) ;
2560:  DO[18181]=((TIMER[9]>=0)) ;
2561:  WAIT ((F[523] AND !F[524]) OR (!F[523] AND F[524]))    ;
2562:  DO[120]=(OFF) ;
2563:  DO[18181]=(OFF) ;
2564:  !WAIT Steuerluft EIN ;
2565:  WAIT ((F[523] AND !F[524] AND DI[2113]) OR (!F[523] AND F[524] AND !DI[2114]) OR (TIMER[9]>=0))    ;
2566:  DO[120]=(TIMER[9]>=0) ;
2567:  DO[18181]=((TIMER[9]>=0)) ;
2568:  WAIT ((F[523] AND !F[524] AND DI[2113]) OR (!F[523] AND F[524] AND !DI[2114]))    ;
2569:  DO[120]=(OFF) ;
2570:  DO[18181]=(OFF) ;
2571:  !In Arbeitsstellung schwenken ;
2572:  DO[2115]=(OFF) ;
2573:  DO[2116]=(ON) ;
2574:  !Freigabe Bewegung (ON) ;
2575:  DO[2117]=(OFF) ;
2576:  DO[2118]=(ON) ;
2577:  TIMER[9]=((-10)) ;
2578:  !Warte bis Spueleimer in Position ;
2579:  WAIT ((!DI[2115] AND DI[2116]) OR (TIMER[9]>=0))    ;
2580:  DO[120]=(TIMER[9]>=0) ;
2581:  DO[18181]=((TIMER[9]>=0)) ;
2582:  WAIT (!DI[2115] AND DI[2116])    ;
2583:  DO[120]=(OFF) ;
2584:  DO[18181]=(OFF) ;
2585:  F[355]=((!DI[2115] AND DI[2116]) OR (F[837])) ;
2586:  WAIT    .30(sec) ;
2587:  !In Ruhestellung schwenken AUS ;
2588:  DO[2115]=(OFF) ;
2589:  !In Arbeitsstellung schw. AUS ;
2590:  DO[2116]=(OFF) ;
2591:  !Freigabe Bewegung AUS ;
2592:  DO[2118]=(OFF) ;
2593:  TIMER[9]=((-5)) ;
2594:  WAIT ((DI[2118]) OR (DI[2117] AND F[837]) OR (TIMER[9]>=0))    ;
2595:  DO[120]=(TIMER[9]>=0) ;
2596:  DO[18181]=((TIMER[9]>=0)) ;
2597:  WAIT ((DI[2118]) OR (DI[2117] AND F[837]))    ;
2598:  DO[120]=(OFF) ;
2599:  DO[18181]=(OFF) ;
2600:  !Freigabe  in  Endlage  halten ;
2601:  DO[2117]=(!F[837]) ;
2602:  IF (F[837]),DO[2118]=PULSE,0.5sec ;
2603:  TIMER[9]=((-10)) ;
2604:  WAIT ((DI[2117]) OR (DI[2118] AND F[837]) OR (TIMER[9]>=0))    ;
2605:  DO[120]=(TIMER[9]>=0) ;
2606:  DO[18181]=((TIMER[9]>=0)) ;
2607:  WAIT ((DI[2117]) OR (DI[2118] AND F[837]))    ;
2608:  DO[120]=(OFF) ;
2609:  DO[18181]=(OFF) ;
2610:  DO[161]=(OFF) ;
2611:  R[42]=44    ;
2612:  JMP LBL[1] ;
2613:   ;
2614:  !******************************** ;
2615:  !*           Schritt 45 ;
2616:  !*         KL1 Spueleimer ;
2617:  !* (an Pneum. Schwenkeinheit KL1) ;
2618:  !*    KL1 in Ruhest. schwenken ;
2619:  !******************************** ;
2620:   ;
2621:  LBL[45] ;
2622:  R[41]=45    ;
2623:  !RSK gestartet ;
2624:  F[321]=(OFF) ;
2625:  DO[161]=(ON) ;
2626:  !Steuerluft EIN ;
2627:  DO[2113]=(ON) ;
2628:  TIMER[9]=((-2)) ;
2629:  !Warte auf Vorwahl Ventilinsel ;
2630:  WAIT ((F[523] AND !F[524]) OR (!F[523] AND F[524]) OR (TIMER[9]>=0))    ;
2631:  DO[120]=(TIMER[9]>=0) ;
2632:  DO[18181]=((TIMER[9]>=0)) ;
2633:  WAIT ((F[523] AND !F[524]) OR (!F[523] AND F[524]))    ;
2634:  DO[120]=(OFF) ;
2635:  DO[18181]=(OFF) ;
2636:  !Warte bis Steuerluft EIN ;
2637:  WAIT ((F[523] AND !F[524] AND DI[2113]) OR (!F[523] AND F[524] AND !DI[2114]) OR (TIMER[9]>=0))    ;
2638:  DO[120]=(TIMER[9]>=0) ;
2639:  DO[18181]=((TIMER[9]>=0)) ;
2640:  WAIT ((F[523] AND !F[524] AND DI[2113]) OR (!F[523] AND F[524] AND !DI[2114]))    ;
2641:  DO[120]=(OFF) ;
2642:  DO[18181]=(OFF) ;
2643:  !In Ruhestellung schwenken EIN ;
2644:  DO[2115]=(ON) ;
2645:  DO[2116]=(OFF) ;
2646:  !Freigabe Bewegung EIN ;
2647:  DO[2117]=(OFF) ;
2648:  DO[2118]=(ON) ;
2649:  TIMER[9]=((-10)) ;
2650:  !Warte bis Spueleimer in Position ;
2651:  WAIT ((DI[2115] AND !DI[2116]) OR (TIMER[9]>=0))    ;
2652:  DO[120]=(TIMER[9]>=0) ;
2653:  DO[18181]=((TIMER[9]>=0)) ;
2654:  WAIT (DI[2115] AND !DI[2116])    ;
2655:  DO[120]=(OFF) ;
2656:  DO[18181]=(OFF) ;
2657:  F[355]=((DI[2115] AND !DI[2116]) OR (F[837])) ;
2658:  WAIT    .30(sec) ;
2659:  !In Ruhestellung schwenken AUS ;
2660:  DO[2115]=(OFF) ;
2661:  !In Arbeitsstellung schw. AUS ;
2662:  DO[2116]=(OFF) ;
2663:  !Freigabe Bewegung AUS ;
2664:  DO[2118]=(OFF) ;
2665:  TIMER[9]=((-5)) ;
2666:  WAIT ((DI[2118]) OR (DI[2117] AND F[837]) OR (TIMER[9]>=0))    ;
2667:  DO[120]=(TIMER[9]>=0) ;
2668:  DO[18181]=((TIMER[9]>=0)) ;
2669:  WAIT ((DI[2118]) OR (DI[2117] AND F[837]))    ;
2670:  DO[120]=(OFF) ;
2671:  DO[18181]=(OFF) ;
2672:  !Freigabe  in  Endlage  halten ;
2673:  DO[2117]=(!F[837]) ;
2674:  IF (F[837]),DO[2118]=PULSE,0.5sec ;
2675:  TIMER[9]=((-10)) ;
2676:  WAIT ((DI[2117]) OR (DI[2118] AND F[837]) OR (TIMER[9]>=0))    ;
2677:  DO[120]=(TIMER[9]>=0) ;
2678:  DO[18181]=((TIMER[9]>=0)) ;
2679:  WAIT ((DI[2117]) OR (DI[2118] AND F[837]))    ;
2680:  DO[120]=(OFF) ;
2681:  DO[18181]=(OFF) ;
2682:  DO[161]=(OFF) ;
2683:  R[42]=45    ;
2684:  JMP LBL[1] ;
2685:   ;
2686:  !******************************** ;
2687:  !*            Schritt 46 ;
2688:  !*          KL2 Spueleimer ;
2689:  !*  (an Pneum. Schwenkeinheit KL2 ;
2690:  !*     KL2 in Arbeitsst. schwenke ;
2691:  !******************************** ;
2692:   ;
2693:  LBL[46] ;
2694:  R[41]=46    ;
2695:  !RSK gestartet ;
2696:  F[321]=(OFF) ;
2697:  DO[177]=(ON) ;
2698:  !Steuerluft EIN ;
2699:  DO[2121]=(ON) ;
2700:  TIMER[9]=((-2)) ;
2701:  !Warte auf Vorwahl Ventilinsel ;
2702:  WAIT ((F[523] AND !F[524]) OR (!F[523] AND F[524]) OR (TIMER[9]>=0))    ;
2703:  DO[120]=(TIMER[9]>=0) ;
2704:  DO[18181]=((TIMER[9]>=0)) ;
2705:  WAIT ((F[523] AND !F[524]) OR (!F[523] AND F[524]))    ;
2706:  DO[120]=(OFF) ;
2707:  DO[18181]=(OFF) ;
2708:  !Warte Steuerluft EIN ;
2709:  WAIT ((F[523] AND !F[524] AND DI[2121]) OR (!F[523] AND F[524] AND !DI[2122]) OR (TIMER[9]>=0))    ;
2710:  DO[120]=(TIMER[9]>=0) ;
2711:  DO[18181]=((TIMER[9]>=0)) ;
2712:  WAIT ((F[523] AND !F[524] AND DI[2121]) OR (!F[523] AND F[524] AND !DI[2122]))    ;
2713:  DO[120]=(OFF) ;
2714:  DO[18181]=(OFF) ;
2715:  !In Arbeitsstellung schwenken EI ;
2716:  DO[2123]=(OFF) ;
2717:  DO[2124]=(ON) ;
2718:  !Freigabe Bewegung EIN ;
2719:  DO[2125]=(OFF) ;
2720:  DO[2126]=(ON) ;
2721:  TIMER[9]=((-10)) ;
2722:  !Warte bis Spueleimer in Position ;
2723:  WAIT ((!DI[2123] AND DI[2124]) OR (TIMER[9]>=0))    ;
2724:  DO[120]=(TIMER[9]>=0) ;
2725:  DO[18181]=((TIMER[9]>=0)) ;
2726:  WAIT (!DI[2123] AND DI[2124])    ;
2727:  DO[120]=(OFF) ;
2728:  DO[18181]=(OFF) ;
2729:  F[376]=(!DI[2123] AND DI[2124]) ;
2730:  WAIT    .30(sec) ;
2731:  !In Ruhestellung schwenken AUS ;
2732:  DO[2123]=(OFF) ;
2733:  !In Arbeitsstellung schwenken AU ;
2734:  DO[2124]=(OFF) ;
2735:  !Freigabe Bewegung AUS ;
2736:  DO[2126]=(OFF) ;
2737:  TIMER[9]=((-5)) ;
2738:  WAIT (DI[2126] OR (TIMER[9]>=0))    ;
2739:  DO[120]=(TIMER[9]>=0) ;
2740:  DO[18181]=((TIMER[9]>=0)) ;
2741:  WAIT (DI[2126])    ;
2742:  DO[120]=(OFF) ;
2743:  DO[18181]=(OFF) ;
2744:  !Freigabe  in  Endlage  halten ;
2745:  DO[2125]=(ON) ;
2746:  TIMER[9]=((-10)) ;
2747:  WAIT (DI[2125] OR (TIMER[9]>=0))    ;
2748:  DO[120]=(TIMER[9]>=0) ;
2749:  DO[18181]=((TIMER[9]>=0)) ;
2750:  WAIT (DI[2125])    ;
2751:  DO[120]=(OFF) ;
2752:  DO[18181]=(OFF) ;
2753:  DO[177]=(OFF) ;
2754:  R[42]=46    ;
2755:  JMP LBL[1] ;
2756:   ;
2757:  !******************************** ;
2758:  !*           Schritt 47 ;
2759:  !*         KL2 Spueleimer ;
2760:  !* (an Pneum. Schwenkeinheit KL2) ;
2761:  !*    KL2 in Ruhest. schwenken ;
2762:  !******************************** ;
2763:   ;
2764:  LBL[47] ;
2765:  R[41]=47    ;
2766:  !RSK gestartet ;
2767:  F[321]=(OFF) ;
2768:  DO[177]=(ON) ;
2769:  !Steuerluft EIN ;
2770:  DO[2121]=(ON) ;
2771:  TIMER[9]=((-2)) ;
2772:  !Warte auf Vorwahl Ventilinsel ;
2773:  WAIT ((F[523] AND !F[524]) OR (!F[523] AND F[524]) OR (TIMER[9]>=0))    ;
2774:  DO[120]=(TIMER[9]>=0) ;
2775:  DO[18181]=((TIMER[9]>=0)) ;
2776:  WAIT ((F[523] AND !F[524]) OR (!F[523] AND F[524]))    ;
2777:  DO[120]=(OFF) ;
2778:  DO[18181]=(OFF) ;
2779:  !Warte Steuerluft EIN ;
2780:  WAIT ((F[523] AND !F[524] AND DI[2121]) OR (!F[523] AND F[524] AND !DI[2122]) OR (TIMER[9]>=0))    ;
2781:  DO[120]=(TIMER[9]>=0) ;
2782:  DO[18181]=((TIMER[9]>=0)) ;
2783:  WAIT ((F[523] AND !F[524] AND DI[2121]) OR (!F[523] AND F[524] AND !DI[2122]))    ;
2784:  DO[120]=(OFF) ;
2785:  DO[18181]=(OFF) ;
2786:  !In Ruhestellung schwenken EIN ;
2787:  DO[2123]=(ON) ;
2788:  DO[2124]=(OFF) ;
2789:  !Freigabe Bewegung EIN ;
2790:  DO[2125]=(OFF) ;
2791:  DO[2126]=(ON) ;
2792:  TIMER[9]=((-10)) ;
2793:  !Warte bis Spueleimer in Position ;
2794:  WAIT ((DI[2123] AND !DI[2124]) OR (TIMER[9]>=0))    ;
2795:  DO[120]=(TIMER[9]>=0) ;
2796:  DO[18181]=((TIMER[9]>=0)) ;
2797:  WAIT (DI[2123] AND !DI[2124])    ;
2798:  DO[120]=(OFF) ;
2799:  DO[18181]=(OFF) ;
2800:  F[376]=(DI[2123] AND !DI[2124]) ;
2801:  WAIT    .30(sec) ;
2802:  !In Ruhestellung schwenken AUS ;
2803:  DO[2123]=(OFF) ;
2804:  !In Arbeitsstellung schwenken AU ;
2805:  DO[2124]=(OFF) ;
2806:  !Freigabe Bewegung AUS ;
2807:  DO[2126]=(OFF) ;
2808:  TIMER[9]=((-5)) ;
2809:  WAIT (DI[2126] OR (TIMER[9]>=0))    ;
2810:  DO[120]=(TIMER[9]>=0) ;
2811:  DO[18181]=((TIMER[9]>=0)) ;
2812:  WAIT (DI[2126])    ;
2813:  DO[120]=(OFF) ;
2814:  DO[18181]=(OFF) ;
2815:  !Freigabe  in  Endlage  halten ;
2816:  DO[2125]=(ON) ;
2817:  TIMER[9]=((-10)) ;
2818:  WAIT (DI[2125] OR (TIMER[9]>=0))    ;
2819:  DO[120]=(TIMER[9]>=0) ;
2820:  DO[18181]=((TIMER[9]>=0)) ;
2821:  WAIT (DI[2125])    ;
2822:  DO[120]=(OFF) ;
2823:  DO[18181]=(OFF) ;
2824:  DO[177]=(OFF) ;
2825:  R[42]=47    ;
2826:  JMP LBL[1] ;
2827:   ;
2828:  !******************************** ;
2829:  !*            Schritt 48 ;
2830:  !*          KL3 Spueleimer ;
2831:  !*  (an Pneum. Schwenkeinheit KL3 ;
2832:  !*     KL3 in Arbeitsst. schwenke ;
2833:  !******************************** ;
2834:   ;
2835:  LBL[48] ;
2836:  R[41]=48    ;
2837:  !RSK gestartet ;
2838:  F[321]=(OFF) ;
2839:  DO[193]=(ON) ;
2840:  !Steuerluft EIN ;
2841:  DO[2129]=(ON) ;
2842:  TIMER[9]=((-2)) ;
2843:  !Warte auf Vorwahl Ventilinsel ;
2844:  WAIT ((F[523] AND !F[524]) OR (!F[523] AND F[524]) OR (TIMER[9]>=0))    ;
2845:  DO[120]=(TIMER[9]>=0) ;
2846:  DO[18181]=((TIMER[9]>=0)) ;
2847:  WAIT ((F[523] AND !F[524]) OR (!F[523] AND F[524]))    ;
2848:  DO[120]=(OFF) ;
2849:  DO[18181]=(OFF) ;
2850:  !Warte bis Steuerluft EIN ;
2851:  WAIT ((F[523] AND !F[524] AND DI[2129]) OR (!F[523] AND F[524] AND !DI[2130]) OR (TIMER[9]>=0))    ;
2852:  DO[120]=(TIMER[9]>=0) ;
2853:  DO[18181]=((TIMER[9]>=0)) ;
2854:  WAIT ((F[523] AND !F[524] AND DI[2129]) OR (!F[523] AND F[524] AND !DI[2130]))    ;
2855:  DO[120]=(OFF) ;
2856:  DO[18181]=(OFF) ;
2857:  !In Arbeitsstellung schwenken EI ;
2858:  DO[2131]=(OFF) ;
2859:  DO[2132]=(ON) ;
2860:  !Freigabe Bewegung EIN ;
2861:  DO[2133]=(OFF) ;
2862:  DO[2134]=(ON) ;
2863:  TIMER[9]=((-10)) ;
2864:  !Warte bis Spueleimer in Position ;
2865:  WAIT ((!DI[2131] AND DI[2132]) OR (TIMER[9]>=0))    ;
2866:  DO[120]=(TIMER[9]>=0) ;
2867:  DO[18181]=((TIMER[9]>=0)) ;
2868:  WAIT (!DI[2131] AND DI[2132])    ;
2869:  DO[120]=(OFF) ;
2870:  DO[18181]=(OFF) ;
2871:  F[397]=(!DI[2131] AND DI[2132]) ;
2872:  WAIT    .30(sec) ;
2873:  !In Ruhestellung schwenken AUS ;
2874:  DO[2131]=(OFF) ;
2875:  ! In Arbeitsstellung schwenken A ;
2876:  DO[2132]=(OFF) ;
2877:  !Freigabe Bewegung AUS ;
2878:  DO[2134]=(OFF) ;
2879:  TIMER[9]=((-5)) ;
2880:  WAIT (DI[2134] OR (TIMER[9]>=0))    ;
2881:  DO[120]=(TIMER[9]>=0) ;
2882:  DO[18181]=((TIMER[9]>=0)) ;
2883:  WAIT (DI[2134])    ;
2884:  DO[120]=(OFF) ;
2885:  DO[18181]=(OFF) ;
2886:  !Freigabe  in  Endlage  halten ;
2887:  DO[2133]=(ON) ;
2888:  TIMER[9]=((-10)) ;
2889:  WAIT (DI[2133] OR (TIMER[9]>=0))    ;
2890:  DO[120]=(TIMER[9]>=0) ;
2891:  DO[18181]=((TIMER[9]>=0)) ;
2892:  WAIT (DI[2133])    ;
2893:  DO[120]=(OFF) ;
2894:  DO[18181]=(OFF) ;
2895:  DO[193]=(OFF) ;
2896:  R[42]=48    ;
2897:  JMP LBL[1] ;
2898:   ;
2899:  !******************************** ;
2900:  !*           Schritt 49 ;
2901:  !*         KL3 Spueleimer ;
2902:  !* (an Pneum. Schwenkeinheit KL3) ;
2903:  !*    KL3 in Ruhest. schwenken ;
2904:  !******************************** ;
2905:   ;
2906:  LBL[49] ;
2907:  R[41]=49    ;
2908:  !RSK gestartet ;
2909:  F[321]=(OFF) ;
2910:  DO[193]=(ON) ;
2911:  !Steuerluft EIN ;
2912:  DO[2129]=(ON) ;
2913:  TIMER[9]=((-2)) ;
2914:  !Warte auf Vorwahl Ventilinsel ;
2915:  WAIT ((F[523] AND !F[524]) OR (!F[523] AND F[524]) OR (TIMER[9]>=0))    ;
2916:  DO[120]=(TIMER[9]>=0) ;
2917:  DO[18181]=((TIMER[9]>=0)) ;
2918:  WAIT ((F[523] AND !F[524]) OR (!F[523] AND F[524]))    ;
2919:  DO[120]=(OFF) ;
2920:  DO[18181]=(OFF) ;
2921:  !Warte bis Steuerluft EIN ;
2922:  WAIT ((F[523] AND !F[524] AND DI[2129]) OR (!F[523] AND F[524] AND !DI[2130]) OR (TIMER[9]>=0))    ;
2923:  DO[120]=(TIMER[9]>=0) ;
2924:  DO[18181]=((TIMER[9]>=0)) ;
2925:  WAIT ((F[523] AND !F[524] AND DI[2129]) OR (!F[523] AND F[524] AND !DI[2130]))    ;
2926:  DO[120]=(OFF) ;
2927:  DO[18181]=(OFF) ;
2928:  !In Ruhestellung schwenken EI ;
2929:  DO[2131]=(ON) ;
2930:  DO[2132]=(OFF) ;
2931:  !Freigabe Bewegung EIN ;
2932:  DO[2133]=(OFF) ;
2933:  DO[2134]=(ON) ;
2934:  TIMER[9]=((-10)) ;
2935:  !Warte bis Spueleimer in Position ;
2936:  WAIT ((DI[2131] AND !DI[2132]) OR (TIMER[9]>=0))    ;
2937:  DO[120]=(TIMER[9]>=0) ;
2938:  DO[18181]=((TIMER[9]>=0)) ;
2939:  WAIT (DI[2131] AND DI[2132])    ;
2940:  DO[120]=(OFF) ;
2941:  DO[18181]=(OFF) ;
2942:  F[397]=(DI[2131] AND !DI[2132]) ;
2943:  WAIT    .30(sec) ;
2944:  !In Ruhestellung schwenken AUS ;
2945:  DO[2131]=(OFF) ;
2946:  !In Arbeitsstellung schwenken A ;
2947:  DO[2132]=(OFF) ;
2948:  !Freigabe Bewegung AUS ;
2949:  DO[2134]=(OFF) ;
2950:  TIMER[9]=((-5)) ;
2951:  WAIT (DI[2134] OR (TIMER[9]>=0))    ;
2952:  DO[120]=(TIMER[9]>=0) ;
2953:  DO[18181]=((TIMER[9]>=0)) ;
2954:  WAIT (DI[2134])    ;
2955:  DO[120]=(OFF) ;
2956:  DO[18181]=(OFF) ;
2957:  !Freigabe  in  Endlage  halten ;
2958:  DO[2133]=(ON) ;
2959:  TIMER[9]=((-10)) ;
2960:  WAIT (DI[2133] OR (TIMER[9]>=0))    ;
2961:  DO[120]=(TIMER[9]>=0) ;
2962:  DO[18181]=((TIMER[9]>=0)) ;
2963:  WAIT (DI[2133])    ;
2964:  DO[120]=(OFF) ;
2965:  DO[18181]=(OFF) ;
2966:  DO[193]=(OFF) ;
2967:  R[42]=49    ;
2968:  JMP LBL[1] ;
2969:   ;
2970:   ;
2971:  !********************** ;
2972:  !*    MS1 Reinigung   * ;
2973:  !*     (an Pneum. )   * ;
2974:  !* Schwenkeinheit MS1 * ;
2975:  !********************** ;
2976:   ;
2977:   ;
2978:  !******************************* ;
2979:  !*         Schritt 50          * ;
2980:  !*       MS1 Reinigung         * ;
2981:  !* MS1 in Arbeitsst. schwenken * ;
2982:  !******************************* ;
2983:   ;
2984:  LBL[50] ;
2985:  R[41]=50    ;
2986:  !RSK gestartet ;
2987:  F[321]=(OFF) ;
2988:  F[323]=(OFF) ;
2989:  F[324]=(OFF) ;
2990:  F[329]=(OFF) ;
2991:  !Reinigung MS1 gestartet ;
2992:  !MS bei Reinigung ;
2993:  DO[116]=(ON) ;
2994:  !Reinigung MS1 gestartet ;
2995:  F[604]=(ON) ;
2996:  !Steuerluft EIN ;
2997:  DO[2161]=(ON) ;
2998:  DO[2163]=(OFF) ;
2999:  DO[2164]=(OFF) ;
3000:  DO[2165]=(OFF) ;
3001:  DO[2166]=(OFF) ;
3002:  DO[2167]=(OFF) ;
3003:  DO[2168]=(OFF) ;
3004:  !Ueberwachungszeit Schwenkeinheit ;
3005:  TIMER[8]=((-5)) ;
3006:  !RSK Fehlerausgabe Schwenkeinheit ;
3007:  F[323]=(!DI[2163]) ;
3008:  !RSK Sammelstoerung ;
3009:  F[329]=(F[323]) ;
3010:  !Sprung bei Fehler MS1 schwenken ;
3011:  IF ((DI[26] OR DI[27]) AND F[323]),JMP LBL[50] ;
3012:  WAIT ((!F[323] OR (TIMER[8]>=0)) AND ((F[523] AND !F[524] AND DI[2161]) OR (!F[523] AND F[524] AND !DI[2162])))    ;
3013:  !Schwenkeinheit 1 in Arbeitsstell ;
3014:  DO[2163]=(OFF) ;
3015:  DO[2164]=(!DO[2164]) ;
3016:  !FRG Bewegung EIN ;
3017:  DO[2165]=(OFF) ;
3018:  DO[2166]=(!DI[2164]) ;
3019:  DO[18181]=(ON) ;
3020:  WAIT ((DI[2164] AND !DI[2163]) OR (TIMER[8]>=0))    ;
3021:  DO[18181]=(OFF) ;
3022:  !RSK Fehlerausgabe Schwenkeinheit ;
3023:  F[324]=((!DI[2164] AND (TIMER[8]>=0)) OR F[324]) ;
3024:  !RSK Sammelstoerung ;
3025:  F[329]=(F[324]) ;
3026:  !In Ruhestellung schwenken AUS ;
3027:  DO[2163]=(OFF) ;
3028:  !In Arbeitsstellung schwenken AUS ;
3029:  DO[2164]=(OFF) ;
3030:  !FRG Bewegung AUS ;
3031:  DO[2166]=(OFF) ;
3032:  IF ((DI[26] OR DI[27]) AND F[324]),JMP LBL[50] ;
3033:  IF (!F[324] AND DI[2166]),JMP LBL[51] ;
3034:   ;
3035:  !*************************** ;
3036:  !*      Schritt 51         * ;
3037:  !*  MS1 Versetzeinheit in  * ;
3038:  !*   Arbeitsst. schwenken  * ;
3039:  !*************************** ;
3040:   ;
3041:  LBL[51] ;
3042:  R[41]=51    ;
3043:  !FRG in Endlage halten ein ;
3044:  DO[2165]=(ON) ;
3045:  DO[2164]=(OFF) ;
3046:  DO[2168]=(OFF) ;
3047:  DO[18181]=(ON) ;
3048:  WAIT (!DI[2165])    ;
3049:  DO[18181]=(OFF) ;
3050:  !Ueberwachungszeit Versetzeinheit ;
3051:  TIMER[8]=((-5)) ;
3052:  !Ueberwachungszeit Reinigung ;
3053:  TIMER[9]=((-6)) ;
3054:  !Versetzeinheit  in  Arbeitsst. ;
3055:  DO[2168]=(!DI[2168] AND F[576]) ;
3056:  IF (DO[2168] AND (TIMER[8]>=0) AND (DI[26] OR DI[27])),JMP LBL[51] ;
3057:  IF ((DI[2168] AND F[576]) OR (!DI[2168] AND !F[576])),JMP LBL[52] ;
3058:   ;
3059:   ;
3060:  !*************************** ;
3061:  !*      Schritt 52         * ;
3062:  !* MS1 Reinigung starten   * ;
3063:  !*************************** ;
3064:   ;
3065:  LBL[52] ;
3066:  R[41]=52    ;
3067:  !MS1 Reinigung i.O. ;
3068:  DO[18181]=(ON) ;
3069:  WAIT (DI[1864])    ;
3070:  DO[18181]=(OFF) ;
3071:  !MS1 Ausblasen EIN ;
3072:  DO[1870]=(ON) ;
3073:  !MS1 Reinigung starten ;
3074:  DO[1864]=(ON) ;
3075:  !Einschaltdauer Reingung ;
3076:  TIMER[7]=((R[26])) ;
3077:  !IF (!DI[1864] AND (TIMER[9]>=0) ;
3078:  DO[18181]=(ON) ;
3079:  WAIT (!DI[1864])    ;
3080:  WAIT ((TIMER[7]>=0))    ;
3081:  DO[18181]=(OFF) ;
3082:  !MS1 Reinigung beenden ;
3083:  DO[1864]=(OFF) ;
3084:  !MS1 Ausblasen AUS ;
3085:  DO[1870]=(OFF) ;
3086:  !MS1 Reinigung i.O. ;
3087:  DO[18181]=(ON) ;
3088:   ;
3089:  WAIT (DI[1864])    ;
3090:  DO[18181]=(OFF) ;
3091:  !MS1 Einspruehen EIN ;
